METHOD FB_init : BOOL
VAR_INPUT
	/// if TRUE, the retain variables are initialized (warm start / cold start)
	bInitRetains: BOOL;
	/// if TRUE, the instance afterwards gets moved into the copy code (online change)
	bInCopyCode: BOOL;
	oid: OTCID;
END_VAR
VAR
	clsId: CLSID;
END_VAR

// initialize flags
bParametersVerified := false;
                    
// set module class id for compatibility check
clsId.Data1 := 16#edbb4036;
clsId.Data2 := 16#240d;
clsId.Data3 := 16#4fd3;
clsId.Data4[0] := 16#9b;
clsId.Data4[1] := 16#53;
clsId.Data4[2] := 16#34;
clsId.Data4[3] := 16#bf;
clsId.Data4[4] := 16#ff;
clsId.Data4[5] := 16#27;
clsId.Data4[6] := 16#d6;
clsId.Data4[7] := 16#ef;

AssignClassId(clsId);
                    
// initialize InitData structure with default values              
stInitData.CallByHdr.indexGroup := 0;
stInitData.CallByHdr.indexOffset := 16#00000000;
stInitData.CallByHdr.cbData := SIZEOF(stInitData.CallBy);
stInitData.CallBy := TctModuleCallByType.Module;
stInitData.ExecutionSequenceHdr.indexGroup := 0;
stInitData.ExecutionSequenceHdr.indexOffset := 16#00000001;
stInitData.ExecutionSequenceHdr.cbData := SIZEOF(stInitData.ExecutionSequence);
stInitData.ExecutionSequence := TctModuleExecutionSequenceType.StateUpdateAfterOutputMapping;
stInitData.StepSizeHdr.indexGroup := 0;
stInitData.StepSizeHdr.indexOffset := 16#00000002;
stInitData.StepSizeHdr.cbData := SIZEOF(stInitData.StepSize);
stInitData.StepSize := TctStepSizeType.UseTaskCycleTime;
stInitData.ExecuteModelCodeHdr.indexGroup := 0;
stInitData.ExecuteModelCodeHdr.indexOffset := 16#00000008;
stInitData.ExecuteModelCodeHdr.cbData := SIZEOF(stInitData.ExecuteModelCode);
stInitData.ExecuteModelCode := 1;
stInitData.ModelParametersHdr.indexGroup := 0;
stInitData.ModelParametersHdr.indexOffset := 16#83000000;
stInitData.ModelParametersHdr.cbData := SIZEOF(stInitData.ModelParameters);
stInitData.ModelParameters.VariableTimeDelay_MaxDelay := 1.00000000000000000e+00;
stInitData.ModelParameters.VariableTimeDelay_InitOutput := 0.00000000000000000e+00;
stInitData.ModelParameters.VariableTimeDelay1_MaxDelay := 1.00000000000000000e+00;
stInitData.ModelParameters.VariableTimeDelay1_InitOutput := 0.00000000000000000e+00;
stInitData.ModelParameters.VariableTimeDelay2_MaxDelay := 1.00000000000000000e+00;
stInitData.ModelParameters.VariableTimeDelay2_InitOutput := 0.00000000000000000e+00;
stInitData.ModelParameters.VariableTimeDelay3_MaxDelay := 1.00000000000000000e+00;
stInitData.ModelParameters.VariableTimeDelay3_InitOutput := 0.00000000000000000e+00;
stInitData.ModelParameters.VariableTimeDelay4_MaxDelay := 1.00000000000000000e+00;
stInitData.ModelParameters.VariableTimeDelay4_InitOutput := 0.00000000000000000e+00;
stInitData.ModelParameters.VariableTimeDelay5_MaxDelay := 1.00000000000000000e+00;
stInitData.ModelParameters.VariableTimeDelay5_InitOutput := 0.00000000000000000e+00;
stInitData.ModelParameters.VariableTimeDelay6_MaxDelay := 1.00000000000000000e+00;
stInitData.ModelParameters.VariableTimeDelay6_InitOutput := 0.00000000000000000e+00;
stInitData.ModelParameters.VariableTimeDelay7_MaxDelay := 1.00000000000000000e+00;
stInitData.ModelParameters.VariableTimeDelay7_InitOutput := 0.00000000000000000e+00;
stInitData.ModelParameters.VariableTimeDelay8_MaxDelay := 1.00000000000000000e+00;
stInitData.ModelParameters.VariableTimeDelay8_InitOutput := 0.00000000000000000e+00;
stInitData.ModelParameters.VariableTimeDelay9_MaxDelay := 1.00000000000000000e+00;
stInitData.ModelParameters.VariableTimeDelay9_InitOutput := 0.00000000000000000e+00;
stInitData.ModelParameters.VariableTimeDelay10_MaxDelay := 1.00000000000000000e+00;
stInitData.ModelParameters.VariableTimeDelay10_InitOutput := 0.00000000000000000e+00;
stInitData.ModelParameters.VariableTimeDelay11_MaxDelay := 1.00000000000000000e+00;
stInitData.ModelParameters.VariableTimeDelay11_InitOutput := 0.00000000000000000e+00;
stInitData.ModelParameters.VariableTimeDelay12_MaxDelay := 1.00000000000000000e+00;
stInitData.ModelParameters.VariableTimeDelay12_InitOutput := 0.00000000000000000e+00;
stInitData.ModelParameters.VariableTimeDelay13_MaxDelay := 1.00000000000000000e+00;
stInitData.ModelParameters.VariableTimeDelay13_InitOutput := 0.00000000000000000e+00;
stInitData.ModelParameters.VariableTimeDelay14_MaxDelay := 1.00000000000000000e+00;
stInitData.ModelParameters.VariableTimeDelay14_InitOutput := 0.00000000000000000e+00;
stInitData.ModelParameters.VariableTimeDelay15_MaxDelay := 1.00000000000000000e+00;
stInitData.ModelParameters.VariableTimeDelay15_InitOutput := 0.00000000000000000e+00;
stInitData.ModelParameters.VariableTimeDelay16_MaxDelay := 1.00000000000000000e+00;
stInitData.ModelParameters.VariableTimeDelay16_InitOutput := 0.00000000000000000e+00;
stInitData.ModelParameters.VariableTimeDelay17_MaxDelay := 1.00000000000000000e+00;
stInitData.ModelParameters.VariableTimeDelay17_InitOutput := 0.00000000000000000e+00;
stInitData.ModelParameters.DataStoreMemory5_InitialValue[0] := 1.00000000000000000e+00;
stInitData.ModelParameters.DataStoreMemory5_InitialValue[1] := 3.00000000000000000e+00;
stInitData.ModelParameters.DataStoreMemory5_InitialValue[2] := 5.00000000000000000e+00;
stInitData.ModelParameters.DataStoreMemory6_InitialValue[0] := 2.00000000000000000e+00;
stInitData.ModelParameters.DataStoreMemory6_InitialValue[1] := 4.00000000000000000e+00;
stInitData.ModelParameters.DataStoreMemory6_InitialValue[2] := 6.00000000000000000e+00;
stInitData.ModelParameters.DataStoreMemory4_InitialValue[0] := 1;
stInitData.ModelParameters.DataStoreMemory4_InitialValue[1] := 0;
stInitData.ModelParameters.DataStoreMemory4_InitialValue[2] := 1;
stInitData.ModelParameters.DataStoreMemory4_InitialValue[3] := 0;
stInitData.ModelParameters.DataStoreMemory4_InitialValue[4] := 1;
stInitData.ModelParameters.DataStoreMemory4_InitialValue[5] := 0;
stInitData.ContextInfoArr_0_TaskOidHdr.indexGroup := 0;
stInitData.ContextInfoArr_0_TaskOidHdr.indexOffset := 16#03002060;
stInitData.ContextInfoArr_0_TaskOidHdr.cbData := SIZEOF(stInitData.ContextInfoArr_0_TaskOid);
stInitData.ContextInfoArr_0_TaskPriorityHdr.indexGroup := 0;
stInitData.ContextInfoArr_0_TaskPriorityHdr.indexOffset := 16#03002070;
stInitData.ContextInfoArr_0_TaskPriorityHdr.cbData := SIZEOF(stInitData.ContextInfoArr_0_TaskPriority);
stInitData.ContextInfoArr_0_TaskCycleTimeNsHdr.indexGroup := 0;
stInitData.ContextInfoArr_0_TaskCycleTimeNsHdr.indexOffset := 16#03002080;
stInitData.ContextInfoArr_0_TaskCycleTimeNsHdr.cbData := SIZEOF(stInitData.ContextInfoArr_0_TaskCycleTimeNs);
stInitData.ContextInfoArr_0_TaskPortHdr.indexGroup := 0;
stInitData.ContextInfoArr_0_TaskPortHdr.indexOffset := 16#03002090;
stInitData.ContextInfoArr_0_TaskPortHdr.cbData := SIZEOF(stInitData.ContextInfoArr_0_TaskPort);
stInitData.ContextInfoArr_0_TaskSortOrderHdr.indexGroup := 0;
stInitData.ContextInfoArr_0_TaskSortOrderHdr.indexOffset := 16#030020b0;
stInitData.ContextInfoArr_0_TaskSortOrderHdr.cbData := SIZEOF(stInitData.ContextInfoArr_0_TaskSortOrder);
stInitData.Header.cbData := SIZEOF(stInitData)-SIZEOF(stInitData.Header);
stInitData.Header.uiElmCnt := 10;


// set pointer to InitData structure
SetInitDataInfo(ADR(stInitData));

// set DataArea information
SetDataAreaInfo(ADR(arrDataAreas),2);
arrDataAreas[1].nDataAreaId := 0;
arrDataAreas[1].nSize := SIZEOF(stInput);
arrDataAreas[1].pPlcVar := ADR(stInput);
arrDataAreas[1].pModuleProcImg := 0;
arrDataAreas[1].eDataAreaType := E_TcMatSimDataAreaType.InputDst;
arrDataAreas[2].nDataAreaId := 1;
arrDataAreas[2].nSize := SIZEOF(stOutput);
arrDataAreas[2].pPlcVar := ADR(stOutput);
arrDataAreas[2].pModuleProcImg := 0;
arrDataAreas[2].eDataAreaType := E_TcMatSimDataAreaType.OutputSrc;


// initialize basic interface pointers and return
FB_init := SUCCEEDED(Init(oid));
END_METHOD

PROPERTY InitData : ST_Tough_Signal_Detection_Simple_InitData
GET
InitData := stInitData;
END_GET
SET
stInitData := InitData;
END_SET
END_PROPERTY

PROPERTY Input_Online : ExtU_Touch_Signal_Detection_S_T
GET
hResult := GetObjPara(16#80000000,sizeof(Input_Online),adr(Input_Online));
END_GET
SET
hResult := SetObjPara(16#80000000,sizeof(Input_Online),adr(Input_Online));
END_SET
END_PROPERTY

{attribute 'object_name' := 'Internal_SetObjState'}
METHOD PROTECTED Internal_SetObjState
VAR_INPUT
	hr: REFERENCE TO HRESULT;
	nextState: TCOM_STATE;
END_VAR

// update pointer to InitData structure
SetInitDataInfo(ADR(stInitData));
// call base method
SUPER^.Internal_SetObjState(hr,nextState);
END_METHOD

PROPERTY MdlInitialized_Online : BOOL
GET
hResult := GetObjPara(16#00000003,sizeof(MdlInitialized_Online),adr(MdlInitialized_Online));
END_GET
SET
hResult := SetObjPara(16#00000003,sizeof(MdlInitialized_Online),adr(MdlInitialized_Online));
END_SET
END_PROPERTY

PROPERTY ModelParameters_Online : P_Touch_Signal_Detection_Simp_T
GET
hResult := GetObjPara(16#83000000,sizeof(ModelParameters_Online),adr(ModelParameters_Online));
END_GET
SET
hResult := SetObjPara(16#83000000,sizeof(ModelParameters_Online),adr(ModelParameters_Online));
END_SET
END_PROPERTY

PROPERTY ModelParameters_Startup : P_Touch_Signal_Detection_Simp_T
GET
ModelParameters_Startup := stInitData.ModelParameters;
END_GET
SET
stInitData.ModelParameters := ModelParameters_Startup;
END_SET
END_PROPERTY

PROPERTY ModuleBuildInfo_Online : TctModuleBuildInfoType
GET
hResult := GetObjPara(16#00000007,sizeof(ModuleBuildInfo_Online),adr(ModuleBuildInfo_Online));
END_GET
SET
hResult := SetObjPara(16#00000007,sizeof(ModuleBuildInfo_Online),adr(ModuleBuildInfo_Online));
END_SET
END_PROPERTY

PROPERTY ModuleInfo_Online : TctModuleInfoType
GET
hResult := GetObjPara(16#00000006,sizeof(ModuleInfo_Online),adr(ModuleInfo_Online));
END_GET
SET
hResult := SetObjPara(16#00000006,sizeof(ModuleInfo_Online),adr(ModuleInfo_Online));
END_SET
END_PROPERTY

{attribute 'object_name' := 'SaveOnlineParametersForInit'}
METHOD SaveOnlineParametersForInit : HRESULT
VAR
	idx: UINT;
	pInitElemHdr: POINTER TO TComInitDataElmHdr;
	pData: PVOID;
	nData: UDINT;
END_VAR
VAR CONSTANT
	nInitDataAlignment: UDINT := 4;
END_VAR

// update pointer to InitData structure
SetInitDataInfo(ADR(stInitData));
// call base method
SaveOnlineParametersForInit := SUPER^.SaveOnlineParametersForInit();
END_METHOD

PROPERTY SimulinkTime_Online : LREAL
GET
hResult := GetObjPara(16#00000005,sizeof(SimulinkTime_Online),adr(SimulinkTime_Online));
END_GET
SET
hResult := SetObjPara(16#00000005,sizeof(SimulinkTime_Online),adr(SimulinkTime_Online));
END_SET
END_PROPERTY

PROPERTY StepSize_Online : TctStepSizeType
GET
hResult := GetObjPara(16#00000002,sizeof(StepSize_Online),adr(StepSize_Online));
END_GET
SET
hResult := SetObjPara(16#00000002,sizeof(StepSize_Online),adr(StepSize_Online));
END_SET
END_PROPERTY

PROPERTY StepSize_Startup : TctStepSizeType
GET
StepSize_Startup := stInitData.StepSize;
END_GET
SET
stInitData.StepSize := StepSize_Startup;
END_SET
END_PROPERTY

{attribute 'object_name' := 'VerifyParameters'}
METHOD PRIVATE VerifyParameters : HRESULT
VAR
	moduleCallByParam: TctModuleCallByType;
END_VAR

IF (bParametersVerified) THEN
  VerifyParameters := Tc2_System.E_HRESULTAdsErr.HRESULT_ADS_NOERROR;
ELSE
  VerifyParameters := GetObjPara(stInitData.CallByHdr.indexOffset,SIZEOF(moduleCallByParam),ADR(moduleCallByParam));
  
  // check the "CallBy" parameter to be set to "Module"
  IF (SUCCEEDED(VerifyParameters) AND (moduleCallByParam <> TctModuleCallByType.Module)) THEN
      VerifyParameters := Tc2_System.E_HRESULTAdsErr.INVALIDPARM;
  END_IF
  
  // set the parameters verified flag
  bParametersVerified := SUCCEEDED(VerifyParameters);
END_IF
END_METHOD

END_FUNCTION_BLOCK

// ---- POUs/Welding_Arm_Movement.TcPOU
PROGRAM Welding_Arm_Movement
VAR_INPUT
	// ===================模块动作信号(按动作先后排列)==========
	Power_Execute 		: BOOL;									// 上电使能控制信号
	Axis_Power			: ARRAY[1..MotorNum] OF BOOL;					// 单电机使能
	Welding_Arm_Power	: BOOL;									// 焊接臂所有电机使能
	
	Home_Execute		: BOOL;									// 设置零点程序使能

	Leg_Home_Set		: ARRAY[1..MotorNum] OF BOOL;	
	Axis_Home_Set		: ARRAY[1..MotorNum] OF BOOL;					// 单电机设定零点信号
	Welding_Arm_Home_Set		: BOOL;							// 焊接臂所有电机设定零点信号

	
	Move_Absolute_Execute		: BOOL;							// 绝对运动使能信号
	Move_Relative_Execute		: BOOL;							// 相对运动使能信号
	Welding_Arm_Move_Execute	: BOOL;							// 焊接臂运动程序使能	
	Axis_Absolute_Eable			: ARRAY[1..MotorNum] OF BOOL;			// 单电机绝对运动使能信号
	Axis_Relative_Eable			: ARRAY[1..MotorNum] OF BOOL;			// 单电机相对运动使能信号
	Welding_Arm_Absolute_Eable	: ARRAY[1..MotorNum] OF BOOL;			// 焊接臂站立使能信号
	Axis_Move_Absolute_Position	: ARRAY[1..MotorNum] OF LREAL;			// 电机绝对运动位置
	Axis_Move_Relative_Position	: ARRAY[1..MotorNum] OF LREAL;			// 电机相对运动位置			
	
	Reset_Execute		: BOOL;									// 电机驱动重置动作发生使能
	Axis_Reset			: ARRAY[1..MotorNum] OF BOOL;					// 单电机驱动重置信号使能
	Welding_Arm_Reset			: BOOL;							// 焊接臂整体电机驱动重置
	
	ExSetPoint_Execute	: BOOL;							// 机器人外部信号发生使能
	ExtSetPointEnable	: BOOL;							// 外部信号发生信号
	ExtSetPointDisable	: BOOL;							// 外部信号结束信号

END_VAR

VAR_OUTPUT
	Digital_Outputs AT%Q* : DINT;					// 数字输出信号（Link到驱动器中的Digital Outputs）
END_VAR

VAR
// =======================NC轴变量==========================
	Axis_Welding_Arm	: ARRAY[1..MotorNum] OF Axis;					// 定义焊接臂轴参量(可以调整数据上限来调整电机数目)
	Leg_Number			: INT;									// 定义焊接臂腿数
	Axis_Number 		: INT;									// 定义轴数目
	
	// ===================状态监测变量=======================
	Power_Status	: ARRAY[1..MotorNum] OF BOOL;						// 上电监测信号
	Leg_Home_Done	: ARRAY[1..MotorNum] OF BOOL;
	Home_Done		: ARRAY[1..MotorNum] OF BOOL;						// 找零监测信号
	MoveAbsoluteDone: ARRAY[1..MotorNum] OF BOOL;						// 电机绝对运动监测信号
	MoveRelativeDone: ARRAY[1..MotorNum] OF BOOL;						// 电机相对运动监测信号
	
	Welding_Arm_Error		: BOOL;								// 焊接臂电机错误信号
	Axis_Error		: ARRAY[1..MotorNum] OF BOOL;						// 电机错误监测信号
	Axis_ErrorID	: ARRAY[1..MotorNum] OF UDINT;						// 电机错误号码监测信号
	
	Axis_ActPostion	: ARRAY[1..MotorNum] OF LREAL;						// 电机轴实际位置
	Axis_ActVelocity: ARRAY[1..MotorNum] OF LREAL;						// 电机轴实际速度
	Mapping_ActPosition	: Variable_Control_Mapping_Model;		// 电机位置映射
	Motor_ActPosition	: ARRAY[1..MotorNum] OF LREAL;					// Mapping后的电机轴实际位置
	
	Current_Turque_Value  AT%IW0 : ARRAY[1..MotorNum] OF INT ;			// 电流、力矩相关值
	Digital_Inputs  AT%I* : ARRAY[1..MotorNum] OF DINT ;				// 数字输入信号（Link到驱动器中的Digital Inputs）
	
	Home_Switch_value : ARRAY[1..MotorNum] OF BOOL;					// 限位开关真假值
	
	Max_Turque_Value 		: INT ;								// 设置最大找零力矩边界值(机械限位法找零时用来判断运动极限位置)
	Switch_Home_Limit		: ARRAY[1..MotorNum] OF DINT ;				// 找零点时接触开关信号值

	Trigger: BOOL;												// The trigger for profile sensor
	
	LScanCounts			: INT;								// 已完成的激光线轮廓扫描数
	ScanTon				: TON;								// 扫描上升沿计时器
	ScanT				: TIME := T#2000MS;					// 扫描上升沿之后的高电平保持时间
	enableScan			: BOOL;								// 开始激光扫描信号
	Digital_Outputs_16: BOOL;
	
	// ====================Simulink模块相关=====================
	Welding_Arm_Simulink		: FB_WeldingArm6AxisMotion_Control(oid:=16#01010050);	// Simulink模型定义
	
		// -- 输入 --
	t_Interval			: LREAL:=0.001;						// 取样时间间隔，默认为1ms
	t					: LREAL:=0;							// 取样当前时间变量，以0为起点
		// -- 输出 --
	T_ALL				: LREAL:=100;						// Simulink模型运动总时长
	ExSetPoint_Position	: ARRAY[1..6] OF LREAL;				// 外部信号位置

	pos_up: LREAL;
	pos_down: LREAL;
	range_v: LREAL;
	pos_far: LREAL;
	pos_near: LREAL;
	range_h: LREAL;
END_VAR

VAR CONSTANT
	MotorNum			: INT := 6;								// 接入控制的电机数量
	
	LScanStepSize		: LREAL := 5;							// 激光扫描步长（LaserScanStepSize），对应电机转角（测试代码）
	LScanRange			: LREAL := 360;							// 激光扫描范围（LaserScanRange），对应电机总转角（测试代码）
END_VAR

// =======================子程序使能(永久运行)===================
Variable_Monitor();			// 变量监测子程序使能
Logic_Control();			// 逻辑控制子程序使能
Variable_Set();				// 变量设置
Welding_Arm_Action();				// 焊接臂整体运动子程序使能
//Safety();					// 保证丝杠行程和电机速度在规定范围内

// =====================电机驱动重置=============================
IF Reset_Execute THEN
	FOR Axis_Number := 1 TO MotorNum {BY 1} DO
		Axis_Welding_Arm[Axis_Number].Reset(Drive_Reset:= Axis_Reset[Axis_Number]);
	END_FOR
END_IF

// =======================电机上电===============================
IF Power_Execute THEN
	FOR Axis_Number := 1 TO MotorNum {BY 1} DO
		Axis_Welding_Arm[Axis_Number].Power(Axis_Enable:= Axis_Power[Axis_Number]);
	END_FOR
END_IF

// =======================找零程序===============================
IF Home_Execute THEN
	// 如果用模型控制，必须加上下面一句话
	Welding_Arm_Simulink.Execute();	// Simulink模型使能
	FOR Axis_Number := 1 TO MotorNum {BY 1} DO
		//Home_Switch_value[Axis_Number] := Digital_Inputs[Axis_Number].20;		// 试验台电机接近开关标识位
//		IF Axis_Number = 1 THEN
//			Home_Switch_value[Axis_Number] := Digital_Inputs[Axis_Number].18;		// 焊接臂升降电机接近开关(上)标识位
//		ELSIF Axis_Number = 2 THEN
//			Home_Switch_value[Axis_Number] := Digital_Inputs[Axis_Number].18;
//		ELSIF Axis_Number = 3 THEN
			// 加入竖直旋转电机后 Digital_Inputs[2].20 需改为 Digital_Inputs[3].20
//			Home_Switch_value[Axis_Number] := Digital_Inputs[Axis_Number].21;		// 焊接臂径向电机接近开关(靠近电机侧)标识位
//		END_IF

		IF Axis_Number = 3 THEN
			Home_Switch_value[Axis_Number] := Digital_Inputs[Axis_Number].21;		// 焊接臂径向电机接近开关(靠近电机侧)标识位
		ELSE
			Home_Switch_value[Axis_Number] := Digital_Inputs[Axis_Number].18;
		END_IF
		
		Axis_Welding_Arm[Axis_Number].Home_Sensor_Backward(	Drive_Home:= Axis_Home_Set[Axis_Number], 
													Home_Switch := Home_Switch_value[Axis_Number]);
	END_FOR
END_IF

// =======================绝对移动程序===============================
IF Move_Absolute_Execute THEN
	FOR Axis_Number := 1 TO MotorNum {BY 1} DO
		Axis_Welding_Arm[Axis_Number].Move_Absolute(	Drive_Move_Absolute:= Axis_Absolute_Eable[Axis_Number], 
														Absolute_Position:= Axis_Move_Absolute_Position[Axis_Number]);
	END_FOR
END_IF

// =======================相对移动程序===============================
IF Move_Relative_Execute THEN
	FOR Axis_Number := 1 TO MotorNum {BY 1} DO
		Axis_Welding_Arm[Axis_Number].Move_Relative(	Drive_Move_Relative:= Axis_Relative_Eable[Axis_Number], 
														Relative_Position:= Axis_Move_Relative_Position[Axis_Number]);
	END_FOR
END_IF

// =================线激光测量触发信号生成程序===================
ScanTon(IN:= enableScan , PT:= ScanT , Q=> , ET=> );

IF Trigger AND (NOT MoveRelativeDone[1]) AND (NOT Digital_Outputs.16)THEN
	Axis_Relative_Eable[1] := TRUE;
END_IF


IF NOT Axis_Relative_Eable[1] AND Trigger THEN
	enableScan := TRUE;
ELSE
	enableScan := FALSE;
END_IF

IF enableScan THEN
	// 输出一定长度的高电平;
	Digital_Outputs.16 := NOT ScanTon.Q;
	Digital_Outputs_16 := Digital_Outputs.16;
	Axis_Relative_Eable[1] := FALSE;
ELSE
	Digital_Outputs.16 := 0;
END_IF

IF Trigger THEN
	IF LScanCounts < LScanRange/LScanStepSize THEN
		IF MoveRelativeDone[1] THEN
			LScanCounts := LScanCounts + 1;
		END_IF		
	END_IF
ELSE
	Digital_Outputs :=0;
END_IF

IF LScanCounts >= LScanRange/LScanStepSize THEN
	Trigger :=0;
	LScanCounts := 0;
END_IF

// =======================外部信号运动程序=======================
IF ExSetPoint_Execute THEN
	//SetGenerator();			// 使能外部信号发生子程序
	Welding_Arm_Simulink.Execute();	// Simulink模型使能
	FOR Axis_Number := 1 TO MotorNum {BY 1} DO
		Axis_Welding_Arm[Axis_Number].ExtSetPoint(Drive_ExtSetPointEnable:= ExtSetPointEnable, 
											Drive_ExtSetPointDisable:= ExtSetPointDisable, 
											ExSetPosition:= ExSetPoint_Position[Axis_Number]);
	END_FOR
	//	Axis_Welding_Arm[1].ExtSetPoint(Drive_ExtSetPointEnable:= ExtSetPointEnable, 
	//										Drive_ExtSetPointDisable:= ExtSetPointDisable, 
	//										ExSetPosition:= ExSetPoint_Position[1]);
	//	Axis_Welding_Arm[3].ExtSetPoint(Drive_ExtSetPointEnable:= ExtSetPointEnable, 
	//										Drive_ExtSetPointDisable:= ExtSetPointDisable, 
	//										ExSetPosition:= ExSetPoint_Position[3]);
END_IF

ACTION Logic_Control:
// =======================控制逻辑区==========================
// 保证所有的动作拥有合理的先后顺序，优化控制逻辑
// 也防止出现两个或两个以上动作同时进行的情况，保证控制安全

// ===================电机驱动重置逻辑========================
//IF Axis_Error[1] OR Axis_Error[2] OR Axis_Error[3] OR Axis_Error[4] OR Axis_Error[5] OR Axis_Error[6] THEN
//	Welding_Arm_Error := TRUE;
//ELSE
//	Welding_Arm_Error := FALSE;
//END_IF
FOR Axis_Number := 1 TO MotorNum {BY 1} DO
	IF Axis_Error[Axis_Number] THEN
		Welding_Arm_Error := TRUE;
		EXIT;
	END_IF
	Welding_Arm_Error := FALSE;
END_FOR

IF Welding_Arm_Error THEN
	Reset_Execute := TRUE;
ELSIF NOT Welding_Arm_Error THEN
	Reset_Execute := FALSE;
ELSIF NOT Reset_Execute THEN
	FOR Axis_Number := 1 TO MotorNum {BY 1} DO
		Axis_Reset[Axis_Number] := FALSE;
		Axis_Welding_Arm[Axis_Number].Reset(Drive_Reset:= Axis_Reset[Axis_Number]);
	END_FOR
END_IF

// =====================上电程序逻辑==========================
IF NOT Power_Execute THEN
	FOR Axis_Number := 1 TO MotorNum {BY 1} DO
		Axis_Power[Axis_Number] := FALSE;
		Axis_Welding_Arm[Axis_Number].Power(Axis_Enable:= Axis_Power[Axis_Number]);
	END_FOR
END_IF

// =====================找零程序逻辑==========================
IF Home_Execute THEN
	FOR Axis_Number := 1 TO MotorNum {BY 1} DO
		IF Home_Done[Axis_Number] THEN			// 	丝杠到达零点位置后，单电机标零使能位关闭			
			Axis_Home_Set[Axis_Number] := FALSE;	
			Axis_Welding_Arm[Axis_Number].Home_Sensor_Backward(	Drive_Home:= Axis_Home_Set[Axis_Number], 
													Home_Switch := NOT Home_Switch_value[Axis_Number]);
		END_IF
	END_FOR
	Move_Absolute_Execute := FALSE;							// 设定零点时，不能进行其他运动
	//ExSetPoint_Execute :=0;
ELSIF NOT Home_Execute THEN
	FOR Axis_Number := 1 TO MotorNum {BY 1} DO
		//Axis_Start_Back[Axis_Number] :=0;
		Axis_Home_Set[Axis_Number] := FALSE;
	END_FOR
END_IF

// =====================焊接臂绝对运动逻辑==========================
IF Move_Absolute_Execute THEN
	//Absolute_Eable := TRUE;
	Home_Execute := FALSE;							// 运动运动使能时，焊接臂调零必须结束
	//ExSetPoint_Execute :=0;						// 运动运动时，不能进行其他运动
	FOR Axis_Number := 1 TO MotorNum {BY 1} DO
		IF MoveAbsoluteDone[Axis_Number] THEN		// 	丝杠到达设定位置后，单电机绝对运动使能位关闭
			Axis_Absolute_Eable[Axis_Number] := FALSE;
		END_IF
	END_FOR
ELSIF NOT Move_Absolute_Execute THEN							// 运动不使能,轴不能运动
	FOR Axis_Number := 1 TO MotorNum {BY 1} DO
		Axis_Absolute_Eable[Axis_Number] := FALSE;
		Axis_Welding_Arm[Axis_Number].Move_Absolute(  Drive_Move_Absolute:= Axis_Absolute_Eable[Axis_Number], 
													  Absolute_Position:= Axis_Move_Absolute_Position[Axis_Number]);
	END_FOR
END_IF

// =====================焊接臂相对运动逻辑==========================
IF Move_Relative_Execute THEN
	//Relative_Eable := TRUE;
	Home_Execute := FALSE;							// 运动运动使能时，焊接臂调零必须结束
	//ExSetPoint_Execute :=0;						// 运动运动时，不能进行其他运动
	FOR Axis_Number := 1 TO MotorNum {BY 1} DO
		IF MoveRelativeDone[Axis_Number] THEN		// 	丝杠到达设定位置后，单电机相对运动使能位关闭
			Axis_Relative_Eable[Axis_Number] := FALSE;
			Axis_Welding_Arm[Axis_Number].Move_Relative(  Drive_Move_Relative:= Axis_Relative_Eable[Axis_Number], 
													  Relative_Position:= Axis_Move_Relative_Position[Axis_Number]);
		END_IF
	END_FOR
ELSIF NOT Move_Relative_Execute THEN							// 运动不使能,轴不能运动
	FOR Axis_Number := 1 TO MotorNum {BY 1} DO
		Axis_Relative_Eable[Axis_Number] := FALSE;
		Axis_Welding_Arm[Axis_Number].Move_Relative(  Drive_Move_Relative:= Axis_Relative_Eable[Axis_Number], 
													  Relative_Position:= Axis_Move_Relative_Position[Axis_Number]);
	END_FOR
END_IF

// =====================外部信号发生逻辑========================
IF ExSetPoint_Execute THEN
	Home_Execute := FALSE;						// 外部信号发生使能时，机器人调零必须结束
ELSIF NOT ExSetPoint_Execute THEN
	ExtSetPointEnable := 0;						// 外部信号发生不使能时，外部信号不能进入程序
	ExtSetPointDisable :=0;
ELSIF ExtSetPointDisable THEN
	ExtSetPointEnable :=0;						// 外部信号发生停止与外部信号发生开始不能同时进行
END_IF
END_ACTION

ACTION Safety:
// 保证丝杠行程和电机速度在规定范围内

// 如果没在找零，检测到焊接臂升降或径向关节接近开关信号即停止焊接臂上所有电机
IF NOT Home_Execute THEN
	// Digital_Inputs[1].19 为焊接臂升降电机接近开关(下)标识位
	// Digital_Inputs[3].20 为焊接臂径向电机接近开关(远离电机侧)标识位
	IF Digital_Inputs[1].18 OR Digital_Inputs[1].19 OR Digital_Inputs[3].20 OR Digital_Inputs[3].21 THEN
		FOR Axis_Number := 1 TO MotorNum {BY 1} DO
			//Axis_Power[Axis_Number] := FALSE;
		END_FOR
	END_IF
END_IF

//IF Digital_Inputs[1].18 THEN
//	pos_up := Axis_Welding_Arm[1].ActPosition;
//	range_v := pos_down - pos_up;
//	Axis_Power[1] := FALSE;
//END_IF
//IF Digital_Inputs[1].19 THEN
//	pos_down := Axis_Welding_Arm[1].ActPosition;
//	Axis_Move_Relative_Position[1] := -300;
//ELSE
//	Axis_Move_Relative_Position[1] := 200;
//END_IF

//IF Digital_Inputs[2].20 THEN
//	pos_far := Axis_Welding_Arm[2].ActPosition;
//	range_h := pos_far - pos_near;
//	Axis_Power[2] := FALSE;
//END_IF
//IF Digital_Inputs[2].21 THEN
//	pos_near := Axis_Welding_Arm[2].ActPosition;

//	Axis_Move_Relative_Position[2] := 200;
//ELSE
//	Axis_Move_Relative_Position[2] := 3;
//END_IF
END_ACTION

ACTION Variable_Monitor:
// =====================关键数据信号监测======================

// ==============最大力矩设置区(边界控制条件)=================
FOR Axis_Number := 1 TO MotorNum {BY 1} DO
	Axis_Welding_Arm[Axis_Number].Max_Turque_Value := Max_Turque_Value;
END_FOR

// =======================力矩检测区==========================
FOR Axis_Number := 1 TO MotorNum {BY 1} DO
	Axis_Welding_Arm[Axis_Number].Current_Turque_Value := Current_Turque_Value[Axis_Number];
END_FOR

// ====================轴实际位置、速度检测区=======================
FOR Axis_Number := 1 TO MotorNum {BY 1} DO
	Axis_ActPostion[Axis_Number] := Axis_Welding_Arm[Axis_Number].ActPosition;
	Axis_ActVelocity[Axis_Number] := Axis_Welding_Arm[Axis_Number].ActVelocity;
END_FOR

// =======================上电状态检测区======================
FOR Axis_Number := 1 TO MotorNum {BY 1} DO
	Power_Status[Axis_Number] := Axis_Welding_Arm[Axis_Number].State_PowerStatus;
END_FOR

// =======================找零状态检测区======================
FOR Axis_Number := 1 TO MotorNum {BY 1} DO
	Home_Done[Axis_Number] := Axis_Welding_Arm[Axis_Number].State_HomeDone;
END_FOR

// ===================电机绝对运动状态检测区==================
FOR Axis_Number := 1 TO MotorNum {BY 1} DO
	MoveAbsoluteDone[Axis_Number] := Axis_Welding_Arm[Axis_Number].State_MoveAbsoluteDone;
END_FOR

// ===================电机相对运动状态检测区==================
FOR Axis_Number := 1 TO MotorNum {BY 1} DO
	MoveRelativeDone[Axis_Number] := Axis_Welding_Arm[Axis_Number].State_MoveRelativeDone;
END_FOR

// =======================电机错误检测区======================
FOR Axis_Number := 1 TO MotorNum {BY 1} DO
	Axis_Error[Axis_Number] := Axis_Welding_Arm[Axis_Number].Axis_Error;
	Axis_ErrorID[Axis_Number] := Axis_Welding_Arm[Axis_Number].Axis_ErrorID;
END_FOR
END_ACTION

ACTION Variable_Set:
// =======================速度规定区==========================
FOR Axis_Number := 1 TO MotorNum {BY 1} DO							//此时每一个电机的速度都是一样的
	Axis_Welding_Arm[Axis_Number].Home_Velocity 	:= 5;			//找零速度(Axis_Jog中的速度)
	Axis_Welding_Arm[Axis_Number].Move_Relative_Velocity	:=5;	//相对运动速度
END_FOR
IF Home_Execute THEN
	//IF Welding_Arm_Home_Set THEN
	//	Axis_Welding_Arm[1].Move_Absolute_Velocity :=20; Axis_Welding_Arm[2].Move_Absolute_Velocity :=20; Axis_Welding_Arm[3].Move_Absolute_Velocity :=20;
	//	Axis_Welding_Arm[4].Move_Absolute_Velocity :=20; Axis_Welding_Arm[5].Move_Absolute_Velocity :=20; Axis_Welding_Arm[6].Move_Absolute_Velocity :=20;
	FOR Axis_Number := 1 TO MotorNum {BY 1} DO
		Axis_Welding_Arm[Axis_Number].Move_Absolute_Velocity := 5;	//找零之后运动至轨迹起始点的速度
	END_FOR
ELSE
	FOR Axis_Number := 1 TO MotorNum {BY 1} DO
			Axis_Welding_Arm[Axis_Number].Move_Absolute_Velocity	:=10;
	END_FOR
END_IF
	

// =======================绝对运动位置规定区==========================
FOR Axis_Number := 1 TO MotorNum {BY 1} DO
	Axis_Move_Absolute_Position[Axis_Number] := 100;
END_FOR

// =======================相对运动位置规定区==========================
FOR Axis_Number := 1 TO MotorNum {BY 1} DO
//	Axis_Move_Relative_Position[Axis_Number] := 360;
//	Axis_Move_Relative_Position[Axis_Number] := LScanStepSize;
	Axis_Move_Relative_Position[Axis_Number] := -15;
END_FOR

// =====================最大力矩规定区========================
Max_Turque_Value := 1400;

// =====================零位传感器限值规定区========================
//Switch_Home_Limit[1]	:= -64028672;
//Switch_Home_Limit[2]	:= 100000;
//Switch_Home_Limit[3]	:= 100000;
//Switch_Home_Limit[4]	:= 100000;
//Switch_Home_Limit[5]	:= 100000;
//Switch_Home_Limit[6]	:= 100000;
//FOR Axis_Number := 1 TO MotorNum {BY 1} DO
//	Switch_Home_Limit[Axis_Number]	:= -64028672;
//END_FOR

// ============电机设置零点后到达位置规定区================
IF Home_Execute THEN
	FOR Axis_Number := 1 TO MotorNum {BY 1} DO
		//Axis_Welding_Arm[Axis_Number].Home_Absolute_Position := 20;
		
		// 如果电机找零调试结束，用下面的语句进行控制，保证找零后的位置为模型起始点
		Axis_Welding_Arm[Axis_Number].Home_Absolute_Position := ExSetPoint_Position[Axis_Number];
	END_FOR
END_IF

// =================线激光测量参数设置区===================

// ===================程序与模型的变量链接===================

	// -- 输入 -- 
Welding_Arm_Simulink.stInput.t := t;								// 采样时间t与Simulink模型中的采样时间链接

	// -- 输出 -- 
T_ALL := Welding_Arm_Simulink.stOutput.T_ALL;
FOR Axis_Number := 1 TO MotorNum {BY 1} DO
	ExSetPoint_Position[Axis_Number] := Welding_Arm_Simulink.stOutput.Disp_J[Axis_Number-1]; // Simulink中的电机输出位移输入到控制模型
END_FOR
END_ACTION

ACTION Welding_Arm_Action:
// =================焊接臂整体运动命令区======================
// 六足所有电机整体控制

// ====================焊接臂驱动重置=========================
IF Welding_Arm_Reset THEN							// 缺少输入
	IF Reset_Execute THEN
		FOR Axis_Number := 1 TO MotorNum {BY 1} DO
			Axis_Reset[Axis_Number] := TRUE;
			Axis_Welding_Arm[Axis_Number].Reset(Drive_Reset:= Axis_Reset[Axis_Number]);
		END_FOR
	END_IF
END_IF	

// ===================焊接臂所有电机上电======================
IF Welding_Arm_Power THEN	
	IF Power_Execute THEN
		FOR Axis_Number := 1 TO MotorNum {BY 1} DO
			Axis_Power[Axis_Number] := TRUE ;
		END_FOR
	END_IF
END_IF
	
// ===================焊接臂找零程序=======================
IF Welding_Arm_Home_Set THEN				// 标零程序
	//Welding_Arm_Start_Back := FALSE;
	IF Home_Execute THEN
		FOR Axis_Number := 1 TO MotorNum {BY 1} DO
			IF NOT Home_Done[Axis_Number] THEN
				Axis_Home_Set[Axis_Number] := TRUE;
				Axis_Welding_Arm[Axis_Number].Home_Sensor_Backward(	Drive_Home:= Axis_Home_Set[Axis_Number], 
													Home_Switch := NOT Home_Switch_value[Axis_Number]);
			ELSIF Home_Done[Axis_Number] THEN
				Axis_Home_Set[Axis_Number] := FALSE;
				Axis_Welding_Arm[Axis_Number].Home_Sensor_Backward(	Drive_Home:= Axis_Home_Set[Axis_Number], 
													Home_Switch := NOT Home_Switch_value[Axis_Number]);
			END_IF
		END_FOR
	ELSIF NOT Home_Execute THEN
		FOR Axis_Number := 1 TO MotorNum {BY 1} DO
			Axis_Home_Set[Axis_Number] := FALSE;
		END_FOR
	END_IF
ELSIF NOT Welding_Arm_Home_Set AND NOT Home_Execute THEN
	FOR Axis_Number := 1 TO MotorNum {BY 1} DO
		Axis_Home_Set[Axis_Number] := FALSE;
	END_FOR
END_IF

// =====================绝对运动程序===============================
IF Welding_Arm_Move_Execute THEN
	IF Move_Absolute_Execute THEN
		FOR Axis_Number := 1 TO MotorNum {BY 1} DO
			IF MoveAbsoluteDone[Axis_Number] THEN		// 	丝杠到达设定位置后，单电机绝对运动使能位关闭
				Axis_Absolute_Eable[Axis_Number] := FALSE;
			ELSE
				Axis_Absolute_Eable[Axis_Number] := TRUE;
			END_IF
		END_FOR
	END_IF
ELSIF NOT Welding_Arm_Move_Execute AND NOT Move_Absolute_Execute THEN 
	FOR Axis_Number := 1 TO MotorNum {BY 1} DO
		Axis_Absolute_Eable[Axis_Number] := FALSE;
	END_FOR
END_IF

// =====================相对运动程序===============================
IF Welding_Arm_Move_Execute THEN
	IF Move_Relative_Execute THEN
		FOR Axis_Number := 1 TO MotorNum {BY 1} DO
			IF MoveRelativeDone[Axis_Number] THEN		// 	丝杠到达设定位置后，单电机相对运动使能位关闭
				Axis_Relative_Eable[Axis_Number] := FALSE;
			ELSE
				Axis_Relative_Eable[Axis_Number] := TRUE;
			END_IF
		END_FOR
	END_IF
ELSIF NOT Welding_Arm_Move_Execute AND NOT Move_Relative_Execute THEN 
	FOR Axis_Number := 1 TO MotorNum {BY 1} DO
		Axis_Relative_Eable[Axis_Number] := FALSE;
	END_FOR
END_IF

// ======================外部信号发生=========================
IF ExtSetPointEnable THEN	
	//FOR Axis_Number := 1 TO 2 {BY 1} DO
	t := t + t_Interval;
	ExtSetPointDisable := FALSE;
	//END_FOR
END_IF

IF t>=T_ALL THEN
	ExtSetPointEnable := FALSE;
	t:=0;
	ExtSetPointDisable := TRUE;
END_IF
END_ACTION

END_PROGRAM

// ---- DUTs/Welding_Arm_Simulink/FB_WeldingArm6AxisMotion_Control.TcPOU
{attribute 'TcDependOnClassFactory' := 'WeldingArm6AxisMotion_Control'}
FUNCTION_BLOCK FB_WeldingArm6AxisMotion_Control EXTENDS FB_TcMatSimObject
VAR_INPUT
	stInput: ST_WeldingArm6AxisMotion_Control_Input;
END_VAR
VAR_OUTPUT
	stOutput: ST_WeldingArm6AxisMotion_Control_Output;
END_VAR
VAR
	stInitData: ST_WeldingArm6AxisMotion_Control_InitData;
	arrDataAreas: ARRAY[1..2] OF ST_TcMatSimObjectDataAreaInfo;
	bParametersVerified: BOOL;
END_VAR

PROPERTY CallBy_Online : TctModuleCallByType
GET
hResult := GetObjPara(16#00000000,sizeof(CallBy_Online),adr(CallBy_Online));
END_GET
SET
hResult := SetObjPara(16#00000000,sizeof(CallBy_Online),adr(CallBy_Online));
END_SET
END_PROPERTY

PROPERTY CallBy_Startup : TctModuleCallByType
GET
CallBy_Startup := stInitData.CallBy;
END_GET
SET
stInitData.CallBy := CallBy_Startup;
END_SET
END_PROPERTY

PROPERTY ContextInfoArr_0_TaskCycleTimeNs_Online : UDINT
GET
hResult := GetObjPara(16#03002080,sizeof(ContextInfoArr_0_TaskCycleTimeNs_Online),adr(ContextInfoArr_0_TaskCycleTimeNs_Online));
END_GET
SET
hResult := SetObjPara(16#03002080,sizeof(ContextInfoArr_0_TaskCycleTimeNs_Online),adr(ContextInfoArr_0_TaskCycleTimeNs_Online));
END_SET
END_PROPERTY

PROPERTY ContextInfoArr_0_TaskCycleTimeNs_Startup : UDINT
GET
ContextInfoArr_0_TaskCycleTimeNs_Startup := stInitData.ContextInfoArr_0_TaskCycleTimeNs;
END_GET
SET
stInitData.ContextInfoArr_0_TaskCycleTimeNs := ContextInfoArr_0_TaskCycleTimeNs_Startup;
END_SET
END_PROPERTY

PROPERTY ContextInfoArr_0_TaskOid_Online : OTCID
GET
hResult := GetObjPara(16#03002060,sizeof(ContextInfoArr_0_TaskOid_Online),adr(ContextInfoArr_0_TaskOid_Online));
END_GET
SET
hResult := SetObjPara(16#03002060,sizeof(ContextInfoArr_0_TaskOid_Online),adr(ContextInfoArr_0_TaskOid_Online));
END_SET
END_PROPERTY

PROPERTY ContextInfoArr_0_TaskOid_Startup : OTCID
GET
ContextInfoArr_0_TaskOid_Startup := stInitData.ContextInfoArr_0_TaskOid;
END_GET
SET
stInitData.ContextInfoArr_0_TaskOid := ContextInfoArr_0_TaskOid_Startup;
END_SET
END_PROPERTY

PROPERTY ContextInfoArr_0_TaskPort_Online : UINT
GET
hResult := GetObjPara(16#03002090,sizeof(ContextInfoArr_0_TaskPort_Online),adr(ContextInfoArr_0_TaskPort_Online));
END_GET
SET
hResult := SetObjPara(16#03002090,sizeof(ContextInfoArr_0_TaskPort_Online),adr(ContextInfoArr_0_TaskPort_Online));
END_SET
END_PROPERTY

PROPERTY ContextInfoArr_0_TaskPort_Startup : UINT
GET
ContextInfoArr_0_TaskPort_Startup := stInitData.ContextInfoArr_0_TaskPort;
END_GET
SET
stInitData.ContextInfoArr_0_TaskPort := ContextInfoArr_0_TaskPort_Startup;
END_SET
END_PROPERTY

PROPERTY ContextInfoArr_0_TaskPriority_Online : UDINT
GET
hResult := GetObjPara(16#03002070,sizeof(ContextInfoArr_0_TaskPriority_Online),adr(ContextInfoArr_0_TaskPriority_Online));
END_GET
SET
hResult := SetObjPara(16#03002070,sizeof(ContextInfoArr_0_TaskPriority_Online),adr(ContextInfoArr_0_TaskPriority_Online));
END_SET
END_PROPERTY

PROPERTY ContextInfoArr_0_TaskPriority_Startup : UDINT
GET
ContextInfoArr_0_TaskPriority_Startup := stInitData.ContextInfoArr_0_TaskPriority;
END_GET
SET
stInitData.ContextInfoArr_0_TaskPriority := ContextInfoArr_0_TaskPriority_Startup;
END_SET
END_PROPERTY

PROPERTY ContextInfoArr_0_TaskSortOrder_Online : UDINT
GET
hResult := GetObjPara(16#030020b0,sizeof(ContextInfoArr_0_TaskSortOrder_Online),adr(ContextInfoArr_0_TaskSortOrder_Online));
END_GET
SET
hResult := SetObjPara(16#030020b0,sizeof(ContextInfoArr_0_TaskSortOrder_Online),adr(ContextInfoArr_0_TaskSortOrder_Online));
END_SET
END_PROPERTY

PROPERTY ContextInfoArr_0_TaskSortOrder_Startup : UDINT
GET
ContextInfoArr_0_TaskSortOrder_Startup := stInitData.ContextInfoArr_0_TaskSortOrder;
END_GET
SET
stInitData.ContextInfoArr_0_TaskSortOrder := ContextInfoArr_0_TaskSortOrder_Startup;
END_SET
END_PROPERTY

PROPERTY CycleUpdateExecuted_Online : BOOL
GET
hResult := GetObjPara(16#00000004,sizeof(CycleUpdateExecuted_Online),adr(CycleUpdateExecuted_Online));
END_GET
SET
hResult := SetObjPara(16#00000004,sizeof(CycleUpdateExecuted_Online),adr(CycleUpdateExecuted_Online));
END_SET
END_PROPERTY

METHOD Execute : HRESULT

IF (SUCCEEDED(hResult)) THEN
  hResult := VerifyParameters();
END_IF

	// update DataArea information
SetDataAreaInfo(ADR(arrDataAreas),2);
	
	// call base method
Execute := SUPER^.Execute();
END_METHOD

PROPERTY ExecuteModelCode_Online : BOOL
GET
hResult := GetObjPara(16#00000008,sizeof(ExecuteModelCode_Online),adr(ExecuteModelCode_Online));
END_GET
SET
hResult := SetObjPara(16#00000008,sizeof(ExecuteModelCode_Online),adr(ExecuteModelCode_Online));
END_SET
END_PROPERTY

PROPERTY ExecuteModelCode_Startup : BOOL
GET
ExecuteModelCode_Startup := stInitData.ExecuteModelCode;
END_GET
SET
stInitData.ExecuteModelCode := ExecuteModelCode_Startup;
END_SET
END_PROPERTY

PROPERTY ExecutionSequence_Online : TctModuleExecutionSequenceType
GET
hResult := GetObjPara(16#00000001,sizeof(ExecutionSequence_Online),adr(ExecutionSequence_Online));
END_GET
SET
hResult := SetObjPara(16#00000001,sizeof(ExecutionSequence_Online),adr(ExecutionSequence_Online));
END_SET
END_PROPERTY

PROPERTY ExecutionSequence_Startup : TctModuleExecutionSequenceType
GET
ExecutionSequence_Startup := stInitData.ExecutionSequence;
END_GET
SET
stInitData.ExecutionSequence := ExecutionSequence_Startup;
END_SET
END_PROPERTY

METHOD FB_init : BOOL
VAR_INPUT
	/// if TRUE, the retain variables are initialized (warm start / cold start)
	bInitRetains: BOOL;
	/// if TRUE, the instance afterwards gets moved into the copy code (online change)
	bInCopyCode: BOOL;
	oid: OTCID;
END_VAR
VAR
	clsId: CLSID;
END_VAR

// initialize flags
bParametersVerified := false;
                    
// set module class id for compatibility check
clsId.Data1 := 16#412caec1;
clsId.Data2 := 16#7008;
clsId.Data3 := 16#47ed;
clsId.Data4[0] := 16#9b;
clsId.Data4[1] := 16#82;
clsId.Data4[2] := 16#ce;
clsId.Data4[3] := 16#15;
clsId.Data4[4] := 16#e3;
clsId.Data4[5] := 16#d3;
clsId.Data4[6] := 16#23;
clsId.Data4[7] := 16#f9;

AssignClassId(clsId);
                    
// initialize InitData structure with default values              
stInitData.CallByHdr.indexGroup := 0;
stInitData.CallByHdr.indexOffset := 16#00000000;
stInitData.CallByHdr.cbData := SIZEOF(stInitData.CallBy);
stInitData.CallBy := TctModuleCallByType.Module;
stInitData.ExecutionSequenceHdr.indexGroup := 0;
stInitData.ExecutionSequenceHdr.indexOffset := 16#00000001;
stInitData.ExecutionSequenceHdr.cbData := SIZEOF(stInitData.ExecutionSequence);
stInitData.ExecutionSequence := TctModuleExecutionSequenceType.StateUpdateAfterOutputMapping;
stInitData.StepSizeHdr.indexGroup := 0;
stInitData.StepSizeHdr.indexOffset := 16#00000002;
stInitData.StepSizeHdr.cbData := SIZEOF(stInitData.StepSize);
stInitData.StepSize := TctStepSizeType.UseTaskCycleTime;
stInitData.ExecuteModelCodeHdr.indexGroup := 0;
stInitData.ExecuteModelCodeHdr.indexOffset := 16#00000008;
stInitData.ExecuteModelCodeHdr.cbData := SIZEOF(stInitData.ExecuteModelCode);
stInitData.ExecuteModelCode := 1;
stInitData.ModelParametersHdr.indexGroup := 0;
stInitData.ModelParametersHdr.indexOffset := 16#82000000;
stInitData.ModelParametersHdr.cbData := SIZEOF(stInitData.ModelParameters);
stInitData.ModelParameters.tcycle_Value := 5.00000000000000000e+00;
stInitData.ModelParameters.J1rg_Value[0] := 2.00000000000000000e+01;
stInitData.ModelParameters.J1rg_Value[1] := 2.00000000000000000e+02;
stInitData.ModelParameters.J2rg_Value[0] := -2.70000000000000000e+02;
stInitData.ModelParameters.J2rg_Value[1] := 9.00000000000000000e+01;
stInitData.ModelParameters.J3rg_Value[0] := 2.00000000000000000e+01;
stInitData.ModelParameters.J3rg_Value[1] := 1.30000000000000000e+02;
stInitData.ModelParameters.phirg_Value[0] := -3.00000000000000000e+01;
stInitData.ModelParameters.phirg_Value[1] := 3.00000000000000000e+01;
stInitData.ModelParameters.gamarg_Value[0] := 1.50000000000000000e+01;
stInitData.ModelParameters.gamarg_Value[1] := 3.50000000000000000e+01;
stInitData.ContextInfoArr_0_TaskOidHdr.indexGroup := 0;
stInitData.ContextInfoArr_0_TaskOidHdr.indexOffset := 16#03002060;
stInitData.ContextInfoArr_0_TaskOidHdr.cbData := SIZEOF(stInitData.ContextInfoArr_0_TaskOid);
stInitData.ContextInfoArr_0_TaskPriorityHdr.indexGroup := 0;
stInitData.ContextInfoArr_0_TaskPriorityHdr.indexOffset := 16#03002070;
stInitData.ContextInfoArr_0_TaskPriorityHdr.cbData := SIZEOF(stInitData.ContextInfoArr_0_TaskPriority);
stInitData.ContextInfoArr_0_TaskCycleTimeNsHdr.indexGroup := 0;
stInitData.ContextInfoArr_0_TaskCycleTimeNsHdr.indexOffset := 16#03002080;
stInitData.ContextInfoArr_0_TaskCycleTimeNsHdr.cbData := SIZEOF(stInitData.ContextInfoArr_0_TaskCycleTimeNs);
stInitData.ContextInfoArr_0_TaskPortHdr.indexGroup := 0;
stInitData.ContextInfoArr_0_TaskPortHdr.indexOffset := 16#03002090;
stInitData.ContextInfoArr_0_TaskPortHdr.cbData := SIZEOF(stInitData.ContextInfoArr_0_TaskPort);
stInitData.ContextInfoArr_0_TaskSortOrderHdr.indexGroup := 0;
stInitData.ContextInfoArr_0_TaskSortOrderHdr.indexOffset := 16#030020b0;
stInitData.ContextInfoArr_0_TaskSortOrderHdr.cbData := SIZEOF(stInitData.ContextInfoArr_0_TaskSortOrder);
stInitData.Header.cbData := SIZEOF(stInitData)-SIZEOF(stInitData.Header);
stInitData.Header.uiElmCnt := 10;


// set pointer to InitData structure
SetInitDataInfo(ADR(stInitData));

// set DataArea information
SetDataAreaInfo(ADR(arrDataAreas),2);
arrDataAreas[1].nDataAreaId := 0;
arrDataAreas[1].nSize := SIZEOF(stInput);
arrDataAreas[1].pPlcVar := ADR(stInput);
arrDataAreas[1].pModuleProcImg := 0;
arrDataAreas[1].eDataAreaType := E_TcMatSimDataAreaType.InputDst;
arrDataAreas[2].nDataAreaId := 1;
arrDataAreas[2].nSize := SIZEOF(stOutput);
arrDataAreas[2].pPlcVar := ADR(stOutput);
arrDataAreas[2].pModuleProcImg := 0;
arrDataAreas[2].eDataAreaType := E_TcMatSimDataAreaType.OutputSrc;


// initialize basic interface pointers and return
FB_init := SUCCEEDED(Init(oid));
END_METHOD

PROPERTY InitData : ST_WeldingArm6AxisMotion_Control_InitData
GET
InitData := stInitData;
END_GET
SET
stInitData := InitData;
END_SET
END_PROPERTY

PROPERTY Input_Online : ExtU_weldingArm6axisMotionTes_T
GET
hResult := GetObjPara(16#80000000,sizeof(Input_Online),adr(Input_Online));
END_GET
SET
hResult := SetObjPara(16#80000000,sizeof(Input_Online),adr(Input_Online));
END_SET
END_PROPERTY

{attribute 'object_name' := 'Internal_SetObjState'}
METHOD PROTECTED Internal_SetObjState
VAR_INPUT
	hr: REFERENCE TO HRESULT;
	nextState: TCOM_STATE;
END_VAR

// update pointer to InitData structure
SetInitDataInfo(ADR(stInitData));
// call base method
SUPER^.Internal_SetObjState(hr,nextState);
END_METHOD

PROPERTY MdlInitialized_Online : BOOL
GET
hResult := GetObjPara(16#00000003,sizeof(MdlInitialized_Online),adr(MdlInitialized_Online));
END_GET
SET
hResult := SetObjPara(16#00000003,sizeof(MdlInitialized_Online),adr(MdlInitialized_Online));
END_SET
END_PROPERTY

PROPERTY ModelParameters_Online : P_weldingArm6axisMotionTest1_T
GET
hResult := GetObjPara(16#82000000,sizeof(ModelParameters_Online),adr(ModelParameters_Online));
END_GET
SET
hResult := SetObjPara(16#82000000,sizeof(ModelParameters_Online),adr(ModelParameters_Online));
END_SET
END_PROPERTY

PROPERTY ModelParameters_Startup : P_weldingArm6axisMotionTest1_T
GET
ModelParameters_Startup := stInitData.ModelParameters;
END_GET
SET
stInitData.ModelParameters := ModelParameters_Startup;
END_SET
END_PROPERTY

PROPERTY ModuleBuildInfo_Online : TctModuleBuildInfoType
GET
hResult := GetObjPara(16#00000007,sizeof(ModuleBuildInfo_Online),adr(ModuleBuildInfo_Online));
END_GET
SET
hResult := SetObjPara(16#00000007,sizeof(ModuleBuildInfo_Online),adr(ModuleBuildInfo_Online));
END_SET
END_PROPERTY

PROPERTY ModuleInfo_Online : TctModuleInfoType
GET
hResult := GetObjPara(16#00000006,sizeof(ModuleInfo_Online),adr(ModuleInfo_Online));
END_GET
SET
hResult := SetObjPara(16#00000006,sizeof(ModuleInfo_Online),adr(ModuleInfo_Online));
END_SET
END_PROPERTY

{attribute 'object_name' := 'SaveOnlineParametersForInit'}
METHOD SaveOnlineParametersForInit : HRESULT
VAR
	idx: UINT;
	pInitElemHdr: POINTER TO TComInitDataElmHdr;
	pData: PVOID;
	nData: UDINT;
END_VAR
VAR CONSTANT
	nInitDataAlignment: UDINT := 4;
END_VAR

// update pointer to InitData structure
SetInitDataInfo(ADR(stInitData));
// call base method
SaveOnlineParametersForInit := SUPER^.SaveOnlineParametersForInit();
END_METHOD

PROPERTY SimulinkTime_Online : LREAL
GET
hResult := GetObjPara(16#00000005,sizeof(SimulinkTime_Online),adr(SimulinkTime_Online));
END_GET
SET
hResult := SetObjPara(16#00000005,sizeof(SimulinkTime_Online),adr(SimulinkTime_Online));
END_SET
END_PROPERTY

PROPERTY StepSize_Online : TctStepSizeType
GET
hResult := GetObjPara(16#00000002,sizeof(StepSize_Online),adr(StepSize_Online));
END_GET
SET
hResult := SetObjPara(16#00000002,sizeof(StepSize_Online),adr(StepSize_Online));
END_SET
END_PROPERTY

PROPERTY StepSize_Startup : TctStepSizeType
GET
StepSize_Startup := stInitData.StepSize;
END_GET
SET
stInitData.StepSize := StepSize_Startup;
END_SET
END_PROPERTY

{attribute 'object_name' := 'VerifyParameters'}
METHOD PRIVATE VerifyParameters : HRESULT
VAR
	moduleCallByParam: TctModuleCallByType;
END_VAR

IF (bParametersVerified) THEN
  VerifyParameters := Tc2_System.E_HRESULTAdsErr.HRESULT_ADS_NOERROR;
ELSE
  VerifyParameters := GetObjPara(stInitData.CallByHdr.indexOffset,SIZEOF(moduleCallByParam),ADR(moduleCallByParam));
  
  // check the "CallBy" parameter to be set to "Module"
  IF (SUCCEEDED(VerifyParameters) AND (moduleCallByParam <> TctModuleCallByType.Module)) THEN
      VerifyParameters := Tc2_System.E_HRESULTAdsErr.INVALIDPARM;
  END_IF
  
  // set the parameters verified flag
  bParametersVerified := SUCCEEDED(VerifyParameters);
END_IF
END_METHOD

END_FUNCTION_BLOCK

// ---- DUTs/Mapping/Leg_Model_Mapping_Control.TcPOU
FUNCTION_BLOCK Leg_Model_Mapping_Control
VAR_INPUT
	Model_Leg		: ARRAY [1..18] OF LREAL;			// 模型中的腿编号
END_VAR
VAR_OUTPUT
	Control_Leg		: ARRAY [1..18] OF LREAL;			// 控制程序中的腿编号
END_VAR

Control_Leg[1] 		:= Model_Leg[1];
Control_Leg[2] 		:= Model_Leg[6];
Control_Leg[3] 		:= Model_Leg[5];
Control_Leg[4] 		:= Model_Leg[4];
Control_Leg[5] 		:= Model_Leg[3];
Control_Leg[6] 		:= Model_Leg[2];

END_FUNCTION_BLOCK

// ---- DUTs/Touch_Signal_Detection/FB_TcMatSimObject_2.TcPOU
FUNCTION_BLOCK FB_TcMatSimObject_2
VAR_INPUT
	/// set this flag to write FB input values to the TcComObject's input DataAreas. This will overwrite the mapped input values before module execution. Set to FALSE to read the mapped input values from the TcComObject to the FB.
	bWriteFbInputValues: BOOL := TRUE;
END_VAR
VAR
	/// process image src and dst pointers and sizes
	pDataAreas: POINTER TO ST_TcMatSimObjectDataAreaInfo;
	nDataAreas: UDINT;
	/// global interface pointers
	ipObjSrv: ITComObjectServer;
	/// object interface pointers
	ipTcComObj: ITComObject;
	ipTcCyclic: ITcCyclic;
	ipTcPostCyclic: ITcPostCyclic;
	ipTcAdi: ITcADI;
	/// task interface pointers
	ipTask: ITcTask;
	/// initial parameters
	pInitData: POINTER TO TComInitDataHdr;
	/// hResult of interface calls (0 if no error)
	hResult: HRESULT;
	/// module class ID
	moduleClsId: CLSID;
	/// expected/desired module class ID
	assignedClsId: CLSID;
	bClassIdVerified: BOOL;
	/// flag indicating whether the module instance was created dynamically
	bDynInstance: BOOL;
	/// the object state at the time FB_init was called, FB_exit will try to switch to this state (only if this means to shift down)
	eInitialObjState: TCOM_STATE := TCOM_STATE.TCOM_STATE_INIT;
END_VAR

METHOD PUBLIC AssignClassId
VAR_INPUT
	clsId : CLSID;
END_VAR
assignedClsId := clsId;
bClassIdVerified := false;
END_METHOD

PROPERTY ClassId : CLSID
GET
hResult := ReadModuleClassId();
ClassId := moduleClsId;
END_GET
END_PROPERTY

PROPERTY Error : BOOL
GET
Error := FAILED(hResult);
END_GET
END_PROPERTY

PROPERTY ErrorCode : HRESULT
GET
ErrorCode := hResult;
END_GET
END_PROPERTY

{attribute 'object_name' := 'Execute'}
METHOD Execute : HRESULT
VAR
	nDaIdx: UDINT;
	pCurDataArea: POINTER TO ST_TcMatSimObjectDataAreaInfo;
END_VAR

IF (SUCCEEDED(hResult)) THEN
  hResult := VerifyClassId();
END_IF

IF (SUCCEEDED(hResult) AND State<>TCOM_STATE_OP) THEN
  hResult := Tc2_System.E_HRESULTAdsErr.NOTREADY;
END_IF

// get image pointers
IF (SUCCEEDED(hResult)) THEN
  GetImagePtrs(hResult);
END_IF

// copy inputs
IF (pDataAreas<>0 AND bWriteFbInputValues) THEN
  FOR nDaIdx:=0 TO nDataAreas-1 DO
    IF (FAILED(hResult))THEN
      CONTINUE;
    END_IF
    pCurDataArea := pDataAreas + nDaIdx*SIZEOF(ST_TcMatSimObjectDataAreaInfo);
    IF ((pCurDataArea^.eDataAreaType <> E_TcMatSimDataAreaType.InputDst))THEN
      CONTINUE;
    END_IF
    IF (pCurDataArea^.pModuleProcImg<>0 AND pCurDataArea^.pPlcVar<>0) THEN
      MEMCPY(pCurDataArea^.pModuleProcImg,pCurDataArea^.pPlcVar,pCurDataArea^.nSize);
    ELSE
      hResult := Tc2_System.E_HRESULTAdsErr.NOINTERFACE;
    END_IF
  END_FOR
END_IF

// call cycle update
IF (SUCCEEDED(hResult)) THEN
  IF (ipTcCyclic<>0) THEN
    hResult := ipTcCyclic.CycleUpdate(ipTask:= ipTask, ipCaller:= 0, context:= 0);
  ELSE
    hResult := Tc2_System.E_HRESULTAdsErr.NOINTERFACE;
  END_IF
END_IF

// copy outputs
IF (pDataAreas<>0) THEN
  FOR nDaIdx:=0 TO nDataAreas-1 DO
    IF (FAILED(hResult))THEN
      CONTINUE;
    END_IF
    pCurDataArea := pDataAreas + nDaIdx*SIZEOF(ST_TcMatSimObjectDataAreaInfo);
    IF ((pCurDataArea^.eDataAreaType = E_TcMatSimDataAreaType.OutputSrc) OR NOT bWriteFbInputValues) THEN
      IF (pCurDataArea^.pModuleProcImg<>0 AND pCurDataArea^.pPlcVar<>0) THEN
        MEMCPY(pCurDataArea^.pPlcVar,pCurDataArea^.pModuleProcImg,pCurDataArea^.nSize);
      ELSE
        hResult := Tc2_System.E_HRESULTAdsErr.NOINTERFACE;
      END_IF
    END_IF
  END_FOR
END_IF


// call post cyclic update
IF (SUCCEEDED(hResult)) THEN
  IF (ipTcPostCyclic<>0) THEN
    hResult := ipTcPostCyclic.PostCyclicUpdate(ipTask:= 0, ipCaller:= 0, context:= 0);
  ELSE
    hResult := Tc2_System.E_HRESULTAdsErr.NOINTERFACE;
  END_IF
END_IF

ReleaseImagePtrs();

Execute := hResult;
END_METHOD

{attribute 'object_name' := 'FB_exit'}
METHOD FB_exit : BOOL
VAR_INPUT
	/// Online Change
	bInCopyCode: BOOL;
END_VAR

IF (NOT bInCopyCode) THEN
  IF (ipObjSrv<>0) THEN
    ipObjSrv.TcRelease();
    ipObjSrv := 0;
  END_IF

  ReleaseTcComInterface();
END_IF
END_METHOD

{attribute 'object_name' := 'FB_init'}
METHOD FB_init : BOOL
VAR_INPUT
	/// init retain variables
	bInitRetains: BOOL;
	/// Online Change
	bInCopyCode: BOOL;
	oid: OTCID;
END_VAR

FB_init := SUCCEEDED(Init(oid));
END_METHOD

{attribute 'object_name' := 'GetImagePtrs'}
METHOD PRIVATE GetImagePtrs
VAR_INPUT
	hr: REFERENCE TO HRESULT;
END_VAR
VAR
	nDaIdx: UDINT;
	pCurDataArea: POINTER TO ST_TcMatSimObjectDataAreaInfo;
END_VAR

IF (ipTcAdi=0) THEN
  hr := Tc2_System.E_HRESULTAdsErr.NOINTERFACE;
END_IF
IF(State<>TCOM_STATE_OP)THEN
  hr := Tc2_System.E_HRESULTAdsErr.INVALIDSTATE;
END_IF


// get pointers to process images
IF (pDataAreas<>0) THEN
  FOR nDaIdx:=0 TO nDataAreas-1 DO
    pCurDataArea := pDataAreas + nDaIdx*SIZEOF(ST_TcMatSimObjectDataAreaInfo);
    IF (FAILED(hr))THEN
      CONTINUE;
    END_IF
    IF ((pCurDataArea^.eDataAreaType <> E_TcMatSimDataAreaType.InputDst) AND (pCurDataArea^.eDataAreaType <> E_TcMatSimDataAreaType.OutputSrc))THEN
      CONTINUE;
    END_IF
    IF (pCurDataArea^.pModuleProcImg=0 AND pCurDataArea^.nSize>0) THEN
      hr := ipTcAdi.GetImagePtr(size:= pCurDataArea^.nSize , offs:=0 , adi_x:=pCurDataArea^.nDataAreaId , ppData:=ADR(pCurDataArea^.pModuleProcImg));
    END_IF
  END_FOR
END_IF

IF (FAILED(hr)) THEN
  ReleaseImagePtrs();
END_IF
END_METHOD

{attribute 'object_name' := 'GetObjPara'}
METHOD GetObjPara : HRESULT
VAR_INPUT
	pid: PTCID;
	nData: UDINT;
	pData: PVOID;
END_VAR

IF (ipTcComObj=0) THEN
  GetObjPara := Tc2_System.E_HRESULTAdsErr.NOINTERFACE;
END_IF

IF (SUCCEEDED(GetObjPara)) THEN
  GetObjPara := ipTcComObj.TcGetObjPara(pid:=pid,nData,pData,0);
END_IF
END_METHOD

{attribute 'object_name' := 'Init'}
METHOD PROTECTED Init : HRESULT
VAR_INPUT
	oid: OTCID;
END_VAR

// preinitialize variables
memset(ADR(moduleClsId),0,SIZEOF(moduleClsId));
bClassIdVerified := FALSE;
hResult := Tc2_System.E_HRESULTAdsErr.HRESULT_ADS_NOERROR;

// get object server
IF (ipObjSrv=0) THEN
  hResult := FW_ObjMgr_GetObjectServer(_AppInfo.ObjId,ADR(ipObjSrv));
END_IF

// try to get object interfaces
IF (SUCCEEDED(hresult)) THEN
  QueryTcComInterface(hResult,oid);
END_IF

// verify class id
IF (SUCCEEDED(hresult)) THEN
  hresult := VerifyClassId();
END_IF

// query interfaces, if the current state is higher than INIT
IF (SUCCEEDED(hresult) AND State>TCOM_STATE.TCOM_STATE_INIT) THEN
  QueryObjInterfaces(hResult);
END_IF

// return value
Init := hresult;
END_METHOD

{attribute 'object_name' := 'InitObjName'}
METHOD PRIVATE InitObjName
VAR_INPUT
	hr: REFERENCE TO HRESULT;
END_VAR
VAR
	objectName: STRING(255) := 'TempContr_PlcRtFbInstance';
	oid: OTCID;
END_VAR

IF (SUCCEEDED(hr)) THEN
  hr := ipTcComObj.TcGetObjectId(oid);
END_IF

IF (SUCCEEDED(hr) and bDynInstance) THEN
  objectName := TC2_STANDARD.CONCAT(objectName,'_');
  objectName := TC2_STANDARD.CONCAT(objectName,UDINT_TO_STRING(oid));
  hr := ipTcComObj.TcSetObjectName(ADR(objectName));
END_IF
END_METHOD

{attribute 'object_name' := 'Internal_SetObjState'}
METHOD PROTECTED Internal_SetObjState
VAR_INPUT
	hr: REFERENCE TO HRESULT;
	nextState: TCOM_STATE;
END_VAR

// verify class id
IF (SUCCEEDED(hr)) THEN
  hr := VerifyClassId();
END_IF

// switch object state
IF (SUCCEEDED(hr) AND nextState>=TCOM_STATE_INIT) THEN
  IF (ipTcComObj=0) THEN
    hr := Tc2_System.E_HRESULTAdsErr.NOINTERFACE;
  END_IF
  IF (ipObjSrv=0) THEN
    hr := Tc2_System.E_HRESULTAdsErr.NOINTERFACE;
  END_IF
  IF (SUCCEEDED(hr)) THEN
    hr := ipTcComObj.TcSetObjState(nextState,ipObjSrv,pInitData);
  END_IF
END_IF
END_METHOD

{attribute 'object_name' := 'QueryObjInterface'}
METHOD PRIVATE QueryObjInterface
VAR_INPUT
	hr: REFERENCE TO HRESULT;
	iid: REFERENCE TO IID;
	pipItf: POINTER TO ITcUnknown;
END_VAR
VAR CONSTANT
	pNull: PVOID := 0;
END_VAR

IF (SUCCEEDED(hr)) THEN
  IF (ipTcComObj=0) THEN
    hr := Tc2_System.E_HRESULTAdsErr.NOINTERFACE;
  ELSIF (pipItf^=ULINT_TO_DWORD(pNull)) THEN
    hr := ipTcComObj.TcQueryInterface(iid:= iid, pipItf:=pipItf);
  END_IF
END_IF
END_METHOD

{attribute 'object_name' := 'QueryObjInterfaces'}
METHOD PRIVATE QueryObjInterfaces
VAR_INPUT
	hr: REFERENCE TO HRESULT;
END_VAR

IF(State<TCOM_STATE_PREOP)THEN
  hr := Tc2_System.E_HRESULTAdsErr.INVALIDSTATE;
END_IF

//cyclic interface
QueryObjInterface(hr,IID_ITCCYCLIC,ADR(ipTcCyclic));
//post cyclic interface
QueryObjInterface(hr,IID_ITCPOSTCYCLIC,ADR(ipTcPostCyclic));
//adi interface
QueryObjInterface(hr,IID_ITcADI,ADR(ipTcAdi));
END_METHOD

{attribute 'object_name' := 'QueryTcComInterface'}
METHOD PRIVATE QueryTcComInterface
VAR_INPUT
	hr: REFERENCE TO HRESULT;
	oid: OTCID;
END_VAR

IF (ipObjSrv=0) THEN
  hr := Tc2_System.E_HRESULTAdsErr.NOINTERFACE;
END_IF

IF (SUCCEEDED(hr) AND ipTcComObj=0) THEN
  bDynInstance := FALSE;
  IF(oid>0) THEN
    // query interface of existing object
    hr := ipObjSrv.TcQueryObjectInterface(oid,IID_ITComObject,ADR(ipTcComObj));
  ELSE
    // create new instance and get the object interface
    hr := ipObjSrv.TcCreateInstance(assignedClsId,IID_ITComObject,ADR(ipTcComObj));
    IF (SUCCEEDED(hr)) THEN
      bDynInstance := TRUE;
      hr := ipTcComObj.TcSetObjectId(OTCID_CreateNewId);
    END_IF
  END_IF
  IF (SUCCEEDED(hr)) THEN
    eInitialObjState := State;
  END_IF
END_IF
END_METHOD

{attribute 'object_name' := 'ReadModuleClassId'}
METHOD PRIVATE ReadModuleClassId : HRESULT
VAR
	emptyClsId: CLSID;
END_VAR
memset(ADR(emptyClsId),0,SIZEOF(emptyClsId));
IF (memcmp(ADR(moduleClsId),ADR(emptyClsId),SIZEOF(moduleClsId))=0) THEN
  IF (ipTcComObj=0) THEN
    ReadModuleClassId := Tc2_System.E_HRESULTAdsErr.NOINTERFACE;
  END_IF

  //objectClsId := clsid;
  IF (SUCCEEDED(ReadModuleClassId)) THEN
    ReadModuleClassId := ipTcComObj.GetClassId(moduleClsId);
  END_IF
END_IF
END_METHOD

{attribute 'object_name' := 'ReleaseImagePtrs'}
METHOD PRIVATE ReleaseImagePtrs : HRESULT
VAR
	nDaIdx: UDINT;
	pCurDataArea: POINTER TO ST_TcMatSimObjectDataAreaInfo;
END_VAR

IF (ipTcAdi=0) THEN
  ReleaseImagePtrs := Tc2_System.E_HRESULTAdsErr.NOINTERFACE;
END_IF

IF (SUCCEEDED(ReleaseImagePtrs) AND pDataAreas<>0) THEN
  // release pointers to the simulink module process images
  FOR nDaIdx:=0 TO nDataAreas-1 DO
    pCurDataArea := pDataAreas + nDaIdx*SIZEOF(ST_TcMatSimObjectDataAreaInfo);

    IF (pCurDataArea^.pModuleProcImg<>0) THEN
      ipTcAdi.ReleaseImagePtr(pData:=pCurDataArea^.pModuleProcImg);
      pCurDataArea^.pModuleProcImg := 0;
    END_IF
  END_FOR
END_IF
END_METHOD

{attribute 'object_name' := 'ReleaseObjInterfaces'}
METHOD PRIVATE ReleaseObjInterfaces : HRESULT

// release interface pointers
IF (ipTcCyclic<>0) THEN
  ipTcCyclic.TcRelease();
  ipTcCyclic := 0;
END_IF
IF (ipTcPostCyclic<>0) THEN
  ipTcPostCyclic.TcRelease();
  ipTcPostCyclic := 0;
END_IF
IF (ipTcAdi<>0) THEN
  ipTcAdi.TcRelease();
  ipTcAdi := 0;
END_IF
END_METHOD

{attribute 'object_name' := 'ReleaseTcComInterface'}
METHOD PRIVATE ReleaseTcComInterface : HRESULT
VAR
	nStateChangeCnt: DINT := 0;
END_VAR

IF (ipTcComObj<>0) THEN
  WHILE (State>eInitialObjState AND nStateChangeCnt<1000) DO
    State := eInitialObjState;
    nStateChangeCnt := nStateChangeCnt+1;
  END_WHILE
  ReleaseObjInterfaces();
  IF (bDynInstance) THEN
    ReleaseTcComInterface := TC3_MODULE.FW_ObjMgr_DeleteInstance(ADR(ipTcComObj));
  ELSE
    ipTcComObj.TcRelease();
  END_IF
  ipTcComObj := 0;
END_IF
END_METHOD

{attribute 'object_name' := 'ResetHresult'}
METHOD ResetHresult
hResult := S_OK;
END_METHOD

{attribute 'object_name' := 'SaveOnlineParametersForInit'}
METHOD SaveOnlineParametersForInit : HRESULT
VAR
	idx: UINT;
	pInitElemHdr: POINTER TO TComInitDataElmHdr;
	pData: PVOID;
	nData: UDINT;
END_VAR
VAR CONSTANT
	nInitDataAlignment: UDINT := 4;
END_VAR
IF (pInitData<>0) THEN
  pInitElemHdr := pInitData + SIZEOF(pInitData^);
  FOR idx:=1 TO pInitData^.uiElmCnt DO
    pData := pInitElemHdr + ULINT_TO_DWORD(SIZEOF(pInitElemHdr^));
    nData := pInitElemHdr^.cbData;
    SaveOnlineParametersForInit := GetObjPara(pInitElemHdr^.indexOffset,nData,pData);
    IF (FAILED(SaveOnlineParametersForInit)) THEN
      RETURN;
    END_IF
    pInitElemHdr := pData + (nInitDataAlignment*((nData + nInitDataAlignment - 1)/nInitDataAlignment));
  END_FOR
ELSE
	SaveOnlineParametersForInit := Tc2_System.E_HRESULTAdsErr.NOTINIT;
END_IF
END_METHOD


METHOD PUBLIC SetDataAreaInfo
VAR_INPUT
  pDataAreas: POINTER TO ST_TcMatSimObjectDataAreaInfo;
  nDataAreas: UDINT;
END_VAR

THIS^.nDataAreas := nDataAreas;
THIS^.pDataAreas := pDataAreas;
END_METHOD


METHOD PUBLIC SetInitDataInfo
VAR_INPUT
  pInitData : POINTER TO TComInitDataHdr;
END_VAR
this^.pInitData := pInitData;
END_METHOD

{attribute 'object_name' := 'SetObjPara'}
METHOD SetObjPara : HRESULT
VAR_INPUT
	pid: PTCID;
	nData: UDINT;
	pData: PVOID;
END_VAR

IF (ipTcComObj=0) THEN
  SetObjPara := Tc2_System.E_HRESULTAdsErr.NOINTERFACE;
END_IF

IF (SUCCEEDED(SetObjPara)) THEN
  SetObjPara := ipTcComObj.TcSetObjPara(pid:=pid,nData,pData,0);
END_IF
END_METHOD

{attribute 'object_name' := 'SetObjState'}
METHOD SetObjState : HRESULT
VAR_INPUT
	finalState: TCOM_STATE;
END_VAR
VAR
	bShiftUp: BOOL;
	bShiftDown: BOOL;
	currentState: TCOM_STATE;
END_VAR

currentState := State;

bShiftUp := finalState>currentState;
bShiftDown := finalState<currentState;

// do not switch up on error
IF (FAILED(hresult)) THEN
  bShiftUp := FALSE;
END_IF
// reset existing error on switching down
IF (bShiftDown) THEN
  ResetHresult();
END_IF

// prepared state switch
CASE currentState OF
  TCOM_STATE_INIT:
    IF(bShiftUp) THEN
      QueryTcComInterface(hResult,0);
      Internal_SetObjState(hResult,TCOM_STATE.TCOM_STATE_PREOP);
      InitObjName(hResult);
    END_IF

  TCOM_STATE_PREOP:
    IF(bShiftUp) THEN
      Internal_SetObjState(hResult,TCOM_STATE.TCOM_STATE_SAFEOP);
      QueryObjInterfaces(hResult);
    ELSIF (bShiftDown) THEN
      Internal_SetObjState(hResult,TCOM_STATE.TCOM_STATE_INIT);
    END_IF

  TCOM_STATE_SAFEOP:
    IF(bShiftUp) THEN
      Internal_SetObjState(hResult,TCOM_STATE.TCOM_STATE_OP);
      QueryObjInterfaces(hResult);
    ELSIF (bShiftDown) THEN
      Internal_SetObjState(hResult,TCOM_STATE.TCOM_STATE_PREOP);
      ReleaseObjInterfaces();
    END_IF


  TCOM_STATE_OP:
    IF (bShiftDown) THEN
      Internal_SetObjState(hResult,TCOM_STATE.TCOM_STATE_SAFEOP);
    END_IF
END_CASE

SetObjState := hResult;
END_METHOD

PROPERTY State : TCOM_STATE
GET
VAR
	hr: HRESULT := S_OK;
	eObjState: TCOM_STATE;
END_VAR

IF (ipTcComObj<>0) THEN
  hr := ipTcComObj.TcGetObjState(ADR(eObjState));
IF (FAILED(hr)) THEN
  eObjState := TCOM_STATE.TCOM_STATE_INIT;
END_IF
ELSE
  eObjState := TCOM_STATE.TCOM_STATE_INIT;
END_IF
State := eObjState;
END_GET
SET
SetObjState(State);
END_SET
END_PROPERTY

{attribute 'object_name' := 'VerifyClassId'}
METHOD PRIVATE VerifyClassId : HRESULT
VAR
	emptyClsId: CLSID;
END_VAR
memset(ADR(emptyClsId),0,SIZEOF(emptyClsId));
IF (bClassIdVerified) THEN
  // class ID was already verified
  VerifyClassId := Tc2_System.E_HRESULTAdsErr.HRESULT_ADS_NOERROR;
ELSIF (memcmp(ADR(assignedClsId),ADR(emptyClsId),SIZEOF(assignedClsId))=0) THEN
  // skip class ID verification if no assignedClsId specified
  VerifyClassId := Tc2_System.E_HRESULTAdsErr.HRESULT_ADS_NOERROR;
ELSE
  // verify class ID
  VerifyClassId := ReadModuleClassId();

  IF (SUCCEEDED(VerifyClassId)) THEN
    IF (memcmp(ADR(assignedClsId),ADR(moduleClsId),SIZEOF(assignedClsId))<>0) THEN
     VerifyClassId := Tc2_System.E_HRESULTAdsErr.INVALIDCLSID;
    END_IF
  END_IF
  bClassIdVerified := SUCCEEDED(VerifyClassId);
END_IF
END_METHOD

END_FUNCTION_BLOCK

// ---- GlobalTextList.TcGTLO
TEXTLIST GlobalTextList
  145 = ' %.2f'
  175 = ' realState=%.3f'
  165 = ' t_Interval=%.2f'
  167 = ' t_Interval=%.3f'
  169 = ' t_Interval=%.4f'
  168 = ' t_Interval=%.5f'
  143 = '%.2f'
  179 = '1'
  81 = 'Axis10_Back'
  82 = 'Axis10_Home'
  117 = 'Axis10_Move'
  11 = 'Axis10_Power'
  83 = 'Axis11_Back'
  84 = 'Axis11_Home'
  118 = 'Axis11_Move'
  12 = 'Axis11_Power'
  85 = 'Axis12_Back'
  86 = 'Axis12_Home'
  119 = 'Axis12_Move'
  13 = 'Axis12_Power'
  87 = 'Axis13_Back'
  88 = 'Axis13_Home'
  120 = 'Axis13_Move'
  14 = 'Axis13_Power'
  89 = 'Axis14_Back'
  90 = 'Axis14_Home'
  121 = 'Axis14_Move'
  15 = 'Axis14_Power'
  91 = 'Axis15_Back'
  92 = 'Axis15_Home'
  122 = 'Axis15_Move'
  16 = 'Axis15_Power'
  93 = 'Axis16_Back'
  94 = 'Axis16_Home'
  123 = 'Axis16_Move'
  17 = 'Axis16_Power'
  95 = 'Axis17_Back'
  96 = 'Axis17_Home'
  124 = 'Axis17_Move'
  18 = 'Axis17_Power'
  97 = 'Axis18_Back'
  98 = 'Axis18_Home'
  125 = 'Axis18_Move'
  19 = 'Axis18_Power'
  62 = 'Axis1_Back'
  64 = 'Axis1_Home'
  63 = 'Axis1_Home_Set'
  106 = 'Axis1_M'
  108 = 'Axis1_Move'
  2 = 'Axis1_Power'
  65 = 'Axis2_Back'
  66 = 'Axis2_Home'
  109 = 'Axis2_Move'
  3 = 'Axis2_Power'
  67 = 'Axis3_Back'
  68 = 'Axis3_Home'
  110 = 'Axis3_Move'
  4 = 'Axis3_Power'
  69 = 'Axis4_Back'
  70 = 'Axis4_Home'
  111 = 'Axis4_Move'
  5 = 'Axis4_Power'
  71 = 'Axis5_Back'
  72 = 'Axis5_Home'
  112 = 'Axis5_Move'
  6 = 'Axis5_Power'
  73 = 'Axis6_Back'
  74 = 'Axis6_Home'
  113 = 'Axis6_Move'
  7 = 'Axis6_Power'
  75 = 'Axis7_Back'
  76 = 'Axis7_Home'
  114 = 'Axis7_Move'
  8 = 'Axis7_Power'
  77 = 'Axis8_Back'
  78 = 'Axis8_Home'
  115 = 'Axis8_Move'
  9 = 'Axis8_Power'
  79 = 'Axis9_Back'
  80 = 'Axis9_Home'
  116 = 'Axis9_Move'
  10 = 'Axis9_Power'
  56 = 'Axis_ActPostion[INDEX]'
  60 = 'Back'
  174 = 'Botton For Step'
  57 = 'Current_Turque_Value[INDEX]'
  39 = 'Driver10_Reset'
  40 = 'Driver11_Reset'
  41 = 'Driver12_Reset'
  42 = 'Driver13_Reset'
  43 = 'Driver14_Reset'
  44 = 'Driver15_Reset'
  45 = 'Driver16_Reset'
  46 = 'Driver17_Reset'
  47 = 'Driver18_Reset'
  30 = 'Driver1_Reset'
  31 = 'Driver2_Reset'
  32 = 'Driver3_Reset'
  33 = 'Driver4_Reset'
  34 = 'Driver5_Reset'
  35 = 'Driver6_Reset'
  36 = 'Driver7_Reset'
  37 = 'Driver8_Reset'
  38 = 'Driver9_Reset'
  127 = 'Error & Reset'
  126 = 'Error&Reset'
  151 = 'Exsetopint_Enable'
  152 = 'Exsetopint_On'
  141 = 'Exsetpoint_Exectue'
  23 = 'Home'
  59 = 'Home_Execute'
  61 = 'Home_Set'
  131 = 'Leg1_Home'
  181 = 'Leg21'
  132 = 'Leg2_Home'
  133 = 'Leg3_Home'
  134 = 'Leg4_Home'
  135 = 'Leg5_Home'
  136 = 'Leg6_Home'
  180 = 'Leg_1'
  186 = 'Leg_16'
  182 = 'Leg_2'
  183 = 'Leg_3'
  184 = 'Leg_4'
  185 = 'Leg_5'
  187 = 'Leg_6'
  177 = 'Model_Position[INDEX]'
  130 = 'Move & Stand'
  107 = 'MoveAbsoluteDone[INDEX]'
  129 = 'Move_Execute'
  53 = 'Power'
  20 = 'Power_Execute'
  188 = 'RealState=%.3f'
  29 = 'Reset'
  49 = 'Reset_Execute'
  26 = 'Robot_Error'
  101 = 'Robot_Home_Set'
  0 = 'Robot_Power'
  48 = 'Robot_Reset'
  128 = 'Robot_Stand_Execute'
  99 = 'Robot_Start_Back'
  100 = 'sadad'
  166 = 'Simulink_Move'
  176 = 'State=%.3f'
  189 = 'Step_Test'
  147 = 't=%.2f'
  170 = 't=%.3f'
  171 = 'Touch_Signal'
  178 = 'Touch_Signal(模型中腿编号)'
  172 = 'Touch_Signal_1'
  173 = 'Touch_Signal_Change'
  144 = 'T_ALL = %.2f'
  158 = 't_Interval=%.2f'
  194 = 'Welding_Arm_Error'
  195 = 'Welding_Arm_Power'
  191 = '上电操作'
  22 = '切换视图'
  157 = '取样时间间隔 t_Interval'
  160 = '取样时间间隔 t_Interval(ms)'
  161 = '取样时间间隔 t_Interval(s)'
  159 = '取样时间间隔 t_Interval/ms'
  139 = '可以用来整体机器人运动'
  140 = '可以用来整体机器人进行Simulink模型验证'
  104 = '可以用来给单个四缸伸长或者是整体机器人站立'
  28 = '可以用来给单个电机或者是整体机器人上电'
  55 = '可以用来给单个电机或者是整体机器人找零'
  103 = '可以用来给单个电机或者是整体机器人站立'
  52 = '可以用来错误时给单个电机或者是整体机器人进行驱动重置'
  24 = '否'
  197 = '复位操作'
  149 = '开始输入轨迹'
  156 = '当前取样时间 t'
  163 = '当前取样时间 t(s)'
  193 = '找零操作'
  25 = '是'
  148 = '是否开始输入轨迹'
  198 = '是否进行Simulink运动操作'
  21 = '是否进行上电操作'
  58 = '是否进行找零操作'
  190 = '是否进行整机上电'
  192 = '是否进行整机找零'
  1 = '是否进行整机操作'
  142 = '是否进行运动操作'
  50 = '是否进行驱动重置'
  199 = '本界面为Welding-Arm操作界面'
  138 = '本界面为电机Sumulink模型运动程序：'
  137 = '本界面为电机Sumulink程序：'
  27 = '本界面为电机上电程序：'
  102 = '本界面为电机伸长/机器人站立程序：'
  54 = '本界面为电机找零程序：'
  105 = '本界面为电机绝对运动/机器人站立程序：'
  201 = '本界面为移动焊机机器人联合控制界面'
  51 = '本界面为驱动重置程序：'
  154 = '输入运动总时长 T_ALL'
  162 = '输入运动总时长 T_ALL(s)'
  150 = '运动当前时间 t'
  164 = '运动当前时间 t(s)'
  146 = '运动总时长 T_ALL'
  196 = '运动总时长 T_ALL(s)'
  200 = '运动操作'
  155 = '运动时间间隔 t'
  153 = '运动终止信号'
END_TEXTLIST

// ---- VISUs/Visu_Home.TcVIS
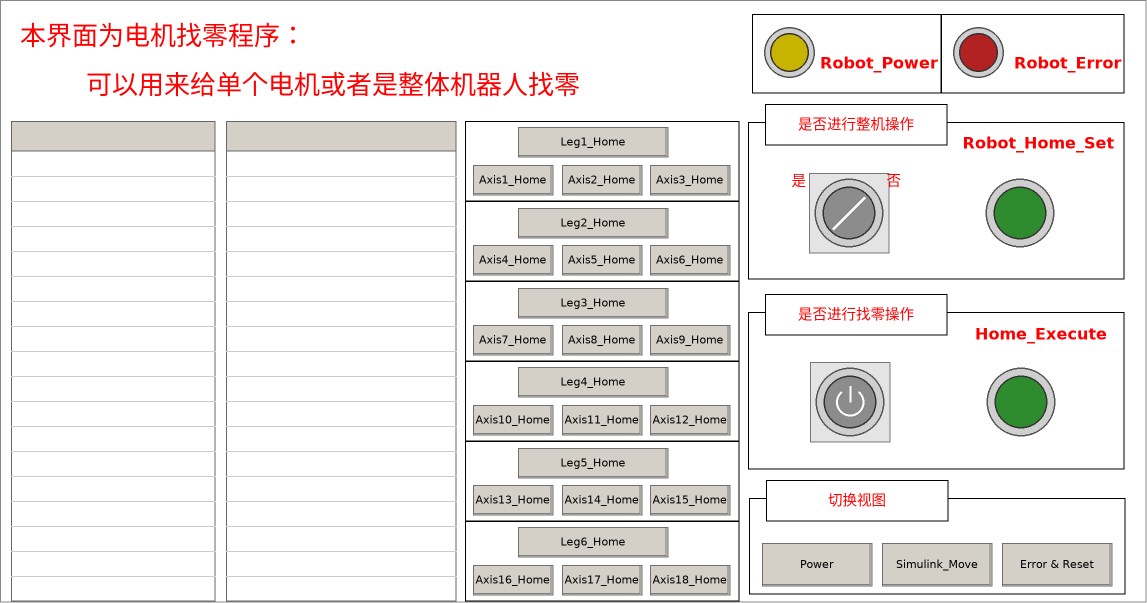
VISUALIZATION Visu_Home  // 1147x603
    Rectangle (752,14 189x79)
    Rectangle (748,312 376x157)
    Label (964,318 154x32), "Home_Execute"
    Rectangle (765,294 182x41), "是否进行找零操作"
    Lamp1 (981,362 80x80), variable: MAIN.Home_Execute, style: Lamp-Lamp1-Green
    PowerSwitch (810,362 80x80), variable: MAIN.Home_Execute, behaviour: TOGGLE, style: Switch-PowerSwitch-Gray
    Rectangle (941,14 183x79)
    Lamp1 (948,23 61x59), variable: MAIN.Robot_Error, style: Lamp-Lamp1-Red
    Label (991,47 154x32), "Robot_Error"
    Label (17,15 365x42), "本界面为电机找零程序："
    Label (83,64 874x42), "可以用来给单个电机或者是整体机器人找零"
    Table (11,121 204x480), data array: MAIN.Axis_ActPostion
        p3854506369: MAIN.Axis_ActPostion[INDEX]
    Table (226,121 230x480), data array: MAIN.Current_Turque_Value
        p3854506369: MAIN.Current_Turque_Value[INDEX]
    Lamp1 (759,23 61x59), variable: MAIN.Robot_Power, style: Lamp-Lamp1-Yellow
    Label (802,47 154x32), "Robot_Power"
    Rectangle (465,121 274x80)
    Button (473,165 80x30), "Axis1_Home"
        toggle MAIN.Axis_Home_Set[1]
        OnMouseClick: change screen: Visu_Home
    Button (650,165 80x30), "Axis3_Home"
        toggle MAIN.Axis_Home_Set[3]
        OnMouseClick: change screen: Visu_Home
    Button (562,165 80x30), "Axis2_Home"
        toggle MAIN.Axis_Home_Set[2]
        OnMouseClick: change screen: Visu_Home
    Rectangle (465,201 274x80)
    Button (473,245 80x30), "Axis4_Home"
        toggle MAIN.Axis_Home_Set[4]
        OnMouseClick: change screen: Visu_Home
    Button (650,245 80x30), "Axis6_Home"
        toggle MAIN.Axis_Home_Set[6]
        OnMouseClick: change screen: Visu_Home
    Button (562,245 80x30), "Axis5_Home"
        toggle MAIN.Axis_Home_Set[5]
        OnMouseClick: change screen: Visu_Home
    Rectangle (465,281 274x80)
    Button (473,325 80x30), "Axis7_Home"
        toggle MAIN.Axis_Home_Set[7]
        OnMouseClick: change screen: Visu_Home
    Button (650,325 80x30), "Axis9_Home"
        toggle MAIN.Axis_Home_Set[9]
        OnMouseClick: change screen: Visu_Home
    Button (562,325 80x30), "Axis8_Home"
        toggle MAIN.Axis_Home_Set[8]
        OnMouseClick: change screen: Visu_Home
    Rectangle (465,361 274x80)
    Button (473,405 80x30), "Axis10_Home"
        toggle MAIN.Axis_Home_Set[10]
        OnMouseClick: change screen: Visu_Home
    Button (650,405 80x30), "Axis12_Home"
        toggle MAIN.Axis_Home_Set[12]
        OnMouseClick: change screen: Visu_Home
    Button (562,405 80x30), "Axis11_Home"
        toggle MAIN.Axis_Home_Set[11]
        OnMouseClick: change screen: Visu_Home
    Rectangle (465,441 274x80)
    Button (473,485 80x30), "Axis13_Home"
        toggle MAIN.Axis_Home_Set[13]
        OnMouseClick: change screen: Visu_Home
    Button (650,485 80x30), "Axis15_Home"
        toggle MAIN.Axis_Home_Set[15]
        OnMouseClick: change screen: Visu_Home
    Button (562,485 80x30), "Axis14_Home"
        toggle MAIN.Axis_Home_Set[14]
        OnMouseClick: change screen: Visu_Home
    Rectangle (465,521 274x80)
    Button (473,565 80x30), "Axis16_Home"
        toggle MAIN.Axis_Home_Set[16]
        OnMouseClick: change screen: Visu_Home
    Button (650,565 80x30), "Axis18_Home"
        toggle MAIN.Axis_Home_Set[18]
        OnMouseClick: change screen: Visu_Home
    Button (562,565 80x30), "Axis17_Home"
        toggle MAIN.Axis_Home_Set[17]
        OnMouseClick: change screen: Visu_Home
    Rectangle (749,498 376x96)
    Rectangle (766,480 182x41), "切换视图"
    Button (762,543 110x43), "Power"
        OnMouseClick: change screen: Visu_Power
    Button (1002,543 110x43), "Error & Reset"
        OnMouseClick: change screen: Visu_Reset
    Button (882,543 110x43), "Simulink_Move"
        OnMouseClick: change screen: Visu_SimulinkMove
    Rectangle (748,122 376x157)
    Rectangle (765,104 182x41), "是否进行整机操作"
    Lamp1 (980,173 80x80), variable: MAIN.Robot_Home_Set, style: Lamp-Lamp1-Green
    RotarySwitch (809,173 80x80), variable: MAIN.Robot_Home_Set, behaviour: TOGGLE, style: Switch-RotarySwitch-Gray
    Label (864,166 60x30), "否"
    Label (769,166 60x30), "是"
    Label (935,127 207x32), "Robot_Home_Set"
    Button (518,127 150x30), "Leg1_Home"
        tap MAIN.Leg_Home_Set[1]
    Button (518,208 150x30), "Leg2_Home"
        tap MAIN.Leg_Home_Set[2]
    Button (518,288 150x30), "Leg3_Home"
        tap MAIN.Leg_Home_Set[3]
    Button (518,367 150x30), "Leg4_Home"
        tap MAIN.Leg_Home_Set[4]
    Button (518,448 150x30), "Leg5_Home"
        tap MAIN.Leg_Home_Set[5]
    Button (518,527 150x30), "Leg6_Home"
        tap MAIN.Leg_Home_Set[6]
END_VISUALIZATION

// ---- VISUs/Visu_Welding_Arm_Move.TcVIS
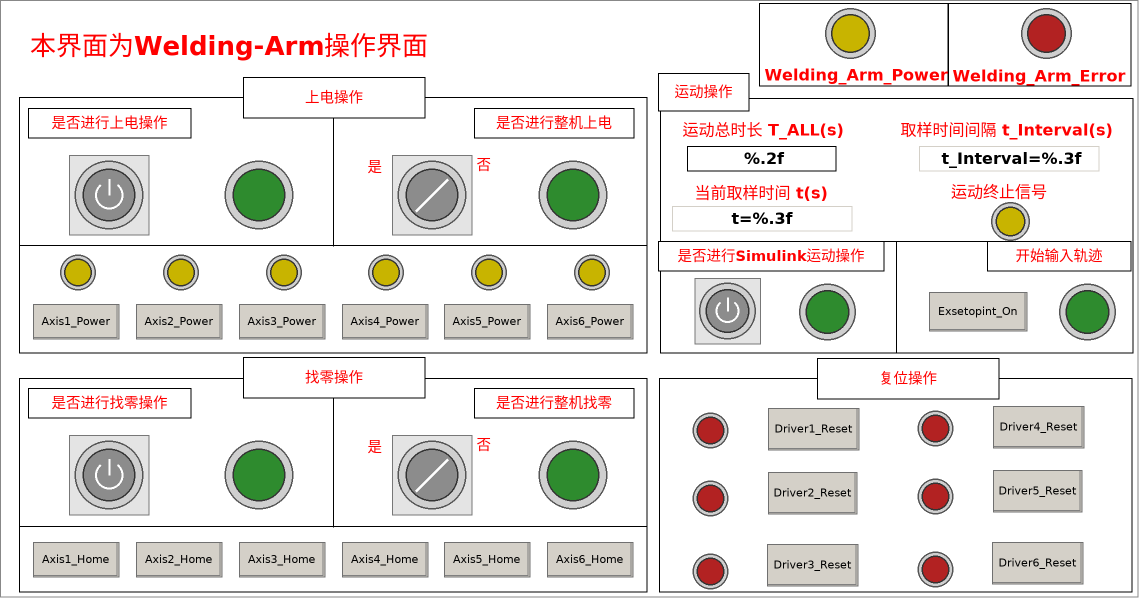
VISUALIZATION Visu_Welding_Arm_Move  // 1139x598
    Rectangle (660,98 473x255)
    Rectangle (659,378 473x214)
    Group (19,97 628x256)
        Rectangle (0,0 628x256)
        Line (1,148) (627,148)
        Line (314,0) (314,149)
    Label (345,152 60x30), "是"
    Label (454,150 60x30), "否"
    Rectangle (474,108 160x30), "是否进行整机上电"
    Lamp1 (219,155 80x80), variable: MAIN.Power_Execute, style: Lamp-Lamp1-Green
    Lamp1 (52,252 52x41), variable: MAIN.Power_Status[1], style: Lamp-Lamp1-Yellow
    Lamp1 (155,252 52x41), variable: MAIN.Power_Status[2], style: Lamp-Lamp1-Yellow
    Lamp1 (258,252 52x41), variable: MAIN.Power_Status[3], style: Lamp-Lamp1-Yellow
    Lamp1 (360,252 52x41), variable: MAIN.Power_Status[4], style: Lamp-Lamp1-Yellow
    Lamp1 (463,252 52x41), variable: MAIN.Power_Status[5], style: Lamp-Lamp1-Yellow
    Lamp1 (566,252 52x41), variable: MAIN.Power_Status[6], style: Lamp-Lamp1-Yellow
    Button (33,304 86x35), "Axis1_Power"
        toggle Welding_Arm_Movement.Axis_Power[1]
    Button (136,304 86x35), "Axis2_Power"
        toggle Welding_Arm_Movement.Axis_Power[2]
    Button (239,304 86x35), "Axis3_Power"
        toggle Welding_Arm_Movement.Axis_Power[3]
    Button (342,304 86x35), "Axis4_Power"
        toggle Welding_Arm_Movement.Axis_Power[4]
    Button (444,304 86x35), "Axis5_Power"
        toggle Welding_Arm_Movement.Axis_Power[5]
    Button (547,304 86x35), "Axis6_Power"
        toggle Welding_Arm_Movement.Axis_Power[6]
    Rectangle (28,108 163x30), "是否进行上电操作"
    PowerSwitch (69,155 80x80), variable: Welding_Arm_Movement.Power_Execute, behaviour: TOGGLE, style: Switch-PowerSwitch-Gray
    Lamp1 (533,155 80x80), variable: MAIN.Robot_Power, style: Lamp-Lamp1-Green
    RotarySwitch (392,155 80x80), variable: Welding_Arm_Movement.Welding_Arm_Power, behaviour: TOGGLE, style: Switch-RotarySwitch-Gray
    Rectangle (243,77 182x41), "上电操作"
    Group (19,378 628x214)
        Rectangle (0,0 628x214)
        Line (1,148) (627,148)
        Line (314,0) (314,149)
    Label (345,432 60x30), "是"
    Label (454,430 60x30), "否"
    Rectangle (474,388 160x30), "是否进行整机找零"
    Lamp1 (219,435 80x80), variable: MAIN.Power_Execute, style: Lamp-Lamp1-Green
    Button (33,542 86x35), "Axis1_Home"
        toggle Welding_Arm_Movement.Axis_Home_Set[1]
    Button (136,542 86x35), "Axis2_Home"
        toggle Welding_Arm_Movement.Axis_Home_Set[2]
    Button (239,542 86x35), "Axis3_Home"
        toggle Welding_Arm_Movement.Axis_Home_Set[3]
    Button (342,542 86x35), "Axis4_Home"
        toggle Welding_Arm_Movement.Axis_Home_Set[4]
    Button (444,542 86x35), "Axis5_Home"
        toggle Welding_Arm_Movement.Axis_Home_Set[5]
    Button (547,542 86x35), "Axis6_Home"
        toggle Welding_Arm_Movement.Axis_Home_Set[6]
    Rectangle (28,388 163x30), "是否进行找零操作"
    PowerSwitch (69,435 80x80), variable: Welding_Arm_Movement.Home_Execute, behaviour: TOGGLE, style: Switch-PowerSwitch-Gray
    Lamp1 (533,435 80x80), variable: MAIN.Robot_Power, style: Lamp-Lamp1-Green
    RotarySwitch (392,435 80x80), variable: Welding_Arm_Movement.Welding_Arm_Home_Set, behaviour: TOGGLE, style: Switch-RotarySwitch-Gray
    Rectangle (243,357 182x41), "找零操作"
    Rectangle (759,3 189x83)
    Rectangle (948,3 183x83)
    Lamp1 (1016,4 61x59), variable: MAIN.Robot_Error, style: Lamp-Lamp1-Red
    Label (953,60 172x32), "Welding_Arm_Error"
    Lamp1 (820,4 61x59), variable: MAIN.Robot_Power, style: Lamp-Lamp1-Yellow
    Label (766,59 181x32), "Welding_Arm_Power"
    Lamp1 (690,406 41x49), variable: Welding_Arm_Movement.Axis_Error[1], style: Lamp-Lamp1-Red
    Lamp1 (690,474 41x49), variable: MAIN.Axis_Error[2], style: Lamp-Lamp1-Red
    Lamp1 (690,547 41x49), variable: MAIN.Axis_Error[3], style: Lamp-Lamp1-Red
    Button (768,408 91x42), "Driver1_Reset"
        tap Welding_Arm_Movement.Axis_Reset[1]
    Button (768,472 89x42), "Driver2_Reset"
        tap Welding_Arm_Movement.Axis_Reset[2]
    Button (767,544 91x42), "Driver3_Reset"
        tap Welding_Arm_Movement.Axis_Reset[3]
    Lamp1 (915,404 41x49), variable: MAIN.Axis_Error[1], style: Lamp-Lamp1-Red
    Lamp1 (915,472 41x49), variable: MAIN.Axis_Error[2], style: Lamp-Lamp1-Red
    Lamp1 (915,545 41x49), variable: MAIN.Axis_Error[3], style: Lamp-Lamp1-Red
    Button (993,406 91x42), "Driver4_Reset"
        tap Welding_Arm_Movement.Axis_Reset[4]
    Button (993,470 89x42), "Driver5_Reset"
        tap Welding_Arm_Movement.Axis_Reset[5]
    Button (992,542 91x42), "Driver6_Reset"
        tap Welding_Arm_Movement.Axis_Reset[6]
    Rectangle (687,146 149x25), "%.2f", text variable: Welding_Arm_Movement.T_ALL
        OnMouseClick: write Robot_Movement.T_ALLWelding_Arm_Movement.T_ALL via Default
    Label (664,118 199x24), "运动总时长 T_ALL(s)"
    Textfield (672,206 180x25), "t=%.3f", text variable: Welding_Arm_Movement.t
    Label (684,181 155x24), "当前取样时间 t(s)"
    Lamp1 (982,199 57x45), variable: Robot_Movement.ExtSetPointDisable, style: Lamp-Lamp1-Yellow
    Label (909,180 180x24), "运动终止信号"
    Label (877,118 260x24), "取样时间间隔 t_Interval(s)"
    Textfield (919,146 180x25), "t_Interval=%.3f", text variable: Welding_Arm_Movement.t_Interval
        OnMouseClick: write Welding_Arm_Movement.t_Interval via Default
    Rectangle (817,358 182x41), "复位操作"
    Line (659,241) (1131,241)
    Rectangle (658,241 226x30), "是否进行Simulink运动操作"
    Lamp1 (791,279 73x66), variable: Robot_Movement.ExSetPoint_Execute, style: Lamp-Lamp1-Green
    PowerSwitch (691,278 73x66), variable: Welding_Arm_Movement.ExSetPoint_Execute, behaviour: TOGGLE, style: Switch-PowerSwitch-Gray
    Rectangle (987,241 144x30), "开始输入轨迹"
    Button (929,292 98x39), "Exsetopint_On"
        toggle Welding_Arm_Movement.ExtSetPointEnable
    Lamp1 (1051,279 73x66), variable: Robot_Movement.ExtSetPointEnable, style: Lamp-Lamp1-Green
    Line (896,242) (896,352)
    Label (27,25 572x42), "本界面为Welding-Arm操作界面"
    Rectangle (658,73 91x38), "运动操作"
END_VISUALIZATION
